//CONTINUE
		//GO_ROBOT:=LOADER_RS4_VAR.I_LOADER_RS4_READY_TAKEUP AND INPUT_G6_VAR.I_G6_READY_PLACING AND INDEXING_2_VAR.O_ROTATION_DONE AND INDEXING_1_VAR.I_INDEXING_1_ROTATION_DONE;
		IF LOADER_RS4_VAR.I_LOADER_RS4_READY_TAKEUP AND INPUT_G6_VAR.I_G6_READY_PLACING AND INDEXING_2_VAR.O_ROTATION_DONE AND INDEXING_1_VAR.I_INDEXING_1_ROTATION_DONE THEN
			GO_ROBOT:=TRUE;
		END_IF
		IF LOADER_RS4_VAR.I_LOADER_RS4_RUNNING AND GO_ROBOT AND NOT LOADER_RS4_VAR.I_LOADER_RS4_READY AND INDEXING_2_VAR.I_INDEXING_2_HOME AND INDEXING_2_VAR.O_ROTATION_DONE THEN
			//TMR3(IN:=GO_ROBOT,PT:=T#0.5S); 
			TMR3(IN:=TRUE,PT:=T#0.5S); 
			POSITION_CHANGED :=FALSE;
		ELSE
			TMR3(IN:=FALSE);
			INDEXING_1_VAR.O_ROTATION_START:=FALSE;	
		END_IF
		LOADER_RS4_VAR.O_LOADER_RS4_CONTINUE :=TMR3.q;
		IF TMR3.Q AND NOT LOADER_RS4_VAR.I_LOADER_RS4_END_CARRIER AND INDEXING_1_VAR.I_INDEXING_1_ROTATION_DONE AND INPUT_VAR.STRAIGHTEN_DONE AND INDEXING_2_VAR.I_INDEXING_2_HOME AND INDEXING_2_VAR.O_ROTATION_DONE  THEN
			IF LOADER_RS4_VAR.LOADER_RS4_OUTPUT_5 <=68  THEN
				POSITION_CHANGED :=TRUE;
			ELSE
				POSITION_CHANGED :=FALSE;
			END_IF	
		END_IF	

		IF ( LOADER_RS4_VAR.I_LOADER_RS4_READY_PLACING OR START_MOVE.Q OR GO_ROBOT)AND NOT LOADER_RS4_VAR.I_LOADER_RS4_READY THEN
			LOADER_RS4_VAR.O_LOADER_RS4_CONTINUE :=TRUE;
		ELSE
			LOADER_RS4_VAR.O_LOADER_RS4_CONTINUE :=FALSE;
		END_IF
	
//END CARRIER		
		IF LOADER_RS4_VAR.LOADER_RS4_OUTPUT_5 >=68 AND LOADER_RS4_VAR.I_LOADER_RS4_READY_TAKEUP THEN
			ROT_START(CLK:=TRUE);
			INDEXING_2_VAR.O_ROTATION_START:=ROT_START.Q;
			//LOADER_RS4_VAR.O_LOADER_RS4_STOP :=ROT_START.Q;
			 RESET_POSITION:=LOADER_RS4_VAR.I_LOADER_RS4_END_CARRIER;
			LOADER_RS4_VAR.I_LOADER_RS4_END_CARRIER:=TRUE;
			ELSE
			ROT_START(CLK:=FALSE);
		END_IF
		
		CNT_INC(CU:=LOADER_RS4_VAR.I_LOADER_RS4_READY_TAKEUP,RESET:= RESET_POSITION,PV:=17);
		LOADER_RS4_VAR.LOADER_RS4_OUTPUT_2:=(WORD_TO_BYTE(CNT_INC.CV)*4)+1 ;
		LOADER_RS4_VAR.LOADER_RS4_OUTPUT_3:=LOADER_RS4_VAR.LOADER_RS4_OUTPUT_2+1 ;
		LOADER_RS4_VAR.LOADER_RS4_OUTPUT_4:=LOADER_RS4_VAR.LOADER_RS4_OUTPUT_3+1 ;
		LOADER_RS4_VAR.LOADER_RS4_OUTPUT_5:=LOADER_RS4_VAR.LOADER_RS4_OUTPUT_4+1 ;
		START_MOVE (IN:=POSITION_CHANGED,PT:=T#0.1S);
	
		IF RESET_POSITION THEN
			RES_POS(IN:=RESET_POSITION,PT:=T#0.5S);
			LOADER_RS4_VAR.LOADER_RS4_OUTPUT_2:=1;
			LOADER_RS4_VAR.LOADER_RS4_OUTPUT_3:=2;
			LOADER_RS4_VAR.LOADER_RS4_OUTPUT_4:=3;
			LOADER_RS4_VAR.LOADER_RS4_OUTPUT_5:=4;
			IF RES_POS.Q THEN
				RESET_POSITION:=FALSE;
				RES_POS(IN:=FALSE);			
			END_IF
		END_IF
		IF NOT SORTER_RS4_VAR.I_SORTER_RS4_ENABLE THEN
			INDEXING_2_VAR.O_ROTATION_START:=LOADER_RS4_VAR.I_LOADER_RS4_END_CARRIER;
		END_IF
			
		CNT_CYCLE(CU:=INDEXING_2_VAR.O_ROTATION_DONE,RESET:=SORTER_RS4_VAR.I_SORTER_RS4_DISABLE,PV:=100);
		IF CNT_CYCLE.CV >=2 THEN
				IF INDEXING_2_VAR.O_ROTATION_DONE THEN
				SORTER_RS4_VAR.I_SORTER_RS4_ENABLE:=TRUE;
			END_IF
		END_IF
		
		IF LOADER_RS4_VAR.I_LOADER_RS4_START_PLACING AND INPUT_G6_VAR.I_G6_START_TAKEUP THEN
			INDEXING_1_VAR.O_ROTATION_START:=TRUE;
			
		END_IF
		IF LOADER_RS4_VAR.I_LOADER_RS4_READY_PLACING THEN
			GO_ROBOT:=FALSE;
		END_IF
		(*
		IF NOT CNT_CYCLE.Q AND LOADER_RS4_VAR.I_LOADER_RS4_END_CYCLE THEN
			START_ROTATE(CLK:=TRUE);
			INDEXING_2_VAR.O_ROTATION_START:= START_ROTATE.Q;	
			ELSE
			START_ROTATE(CLK:=FALSE);
		END_IF
					SORTER_RS4_VAR.I_SORTER_RS4_ENABLE:=TRUE;
		*)
	END_IF
END_IF


ELSE
	LOADER_RS4_VAR.O_LOADER_RS4_STOP:=TRUE;
	IF LOADER_RS4_VAR.I_LOADER_RS4_READY THEN
		LOADER_RS4_VAR.O_LOADER_RS4_SETMOTORON:=FALSE;
	END_IF
END_IF

END_PROGRAM

// ---- POUs/ROBOT/SORTER_RS4.TcPOU
PROGRAM SORTER_RS4
VAR

	TMR10: TON;
	TMR8: TON;
	TMR9: TON;
	TMR7: TON;
	TMR3: TON;
	POSITION_CHANGED: BOOL;
	START_MOVE: TP;
	TMR1: TON;
	TP2: TP;
	START_ROBOT: TP;
	TMR2: TON;
	GO_ROBOT: BOOL;
	TP_COUNT: R_TRIG;
	CNT_INC: CTU;
	VAL: INT;
	ROT_START:R_TRIG;
	RESET_POSITION: BOOL;
	RES_POS: TON;
	STRY_CONTINUE: TP;
END_VAR


IF SORTER_RS4_VAR.I_SORTER_RS4_ENABLE THEN
IF SORTER_RS4_VAR.IX_SORTER_RS4_GRIPPER_1 THEN
	SORTER_RS4_VAR.O_SORTER_RS4_GRIPPER_CLOSE_1:=TRUE;
	SORTER_RS4_VAR.O_SORTER_RS4_GRIPPER_OPEN_1:=FALSE;
ELSE
	SORTER_RS4_VAR.O_SORTER_RS4_GRIPPER_CLOSE_1:=FALSE;
	SORTER_RS4_VAR.O_SORTER_RS4_GRIPPER_OPEN_1:=TRUE;
END_IF

IF SORTER_RS4_VAR.IX_SORTER_RS4_GRIPPER_2 THEN
	SORTER_RS4_VAR.O_SORTER_RS4_GRIPPER_CLOSE_2:=TRUE;
	SORTER_RS4_VAR.O_SORTER_RS4_GRIPPER_OPEN_2:=FALSE;
ELSE
	SORTER_RS4_VAR.O_SORTER_RS4_GRIPPER_CLOSE_2:=FALSE;
	SORTER_RS4_VAR.O_SORTER_RS4_GRIPPER_OPEN_2:=TRUE;
END_IF

IF SORTER_RS4_VAR.IX_SORTER_RS4_GRIPPER_3 THEN
	SORTER_RS4_VAR.O_SORTER_RS4_GRIPPER_CLOSE_3:=TRUE;
	SORTER_RS4_VAR.O_SORTER_RS4_GRIPPER_OPEN_3:=FALSE;
ELSE
	SORTER_RS4_VAR.O_SORTER_RS4_GRIPPER_CLOSE_3:=FALSE;
	SORTER_RS4_VAR.O_SORTER_RS4_GRIPPER_OPEN_3:=TRUE;
END_IF

IF SORTER_RS4_VAR.IX_SORTER_RS4_GRIPPER_4 THEN
	SORTER_RS4_VAR.O_SORTER_RS4_GRIPPER_CLOSE_4:=TRUE;
	SORTER_RS4_VAR.O_SORTER_RS4_GRIPPER_OPEN_4:=FALSE;
ELSE
	SORTER_RS4_VAR.O_SORTER_RS4_GRIPPER_CLOSE_4:=FALSE;
	SORTER_RS4_VAR.O_SORTER_RS4_GRIPPER_OPEN_4:=TRUE;
END_IF

IF SORTER_RS4_VAR.IX_SORTER_RS4_GRIPPER_EXT_1 THEN
	SORTER_RS4_VAR.O_SORTER_RS4_GRIPPER_EXT_DOWN_1:=TRUE;
	SORTER_RS4_VAR.O_SORTER_RS4_GRIPPER_EXT_UP_1:=FALSE;
ELSE
	SORTER_RS4_VAR.O_SORTER_RS4_GRIPPER_EXT_DOWN_1:=FALSE;
	SORTER_RS4_VAR.O_SORTER_RS4_GRIPPER_EXT_UP_1:=TRUE;
END_IF


IF SORTER_RS4_VAR.IX_SORTER_RS4_GRIPPER_EXT_2 THEN
	SORTER_RS4_VAR.O_SORTER_RS4_GRIPPER_EXT_DOWN_2:=TRUE;
	SORTER_RS4_VAR.O_SORTER_RS4_GRIPPER_EXT_UP_2:=FALSE;
ELSE
	SORTER_RS4_VAR.O_SORTER_RS4_GRIPPER_EXT_DOWN_2:=FALSE;
	SORTER_RS4_VAR.O_SORTER_RS4_GRIPPER_EXT_UP_2:=TRUE;
END_IF


IF SORTER_RS4_VAR.IX_SORTER_RS4_GRIPPER_EXT_3 THEN
	SORTER_RS4_VAR.O_SORTER_RS4_GRIPPER_EXT_DOWN_3:=TRUE;
	SORTER_RS4_VAR.O_SORTER_RS4_GRIPPER_EXT_UP_3:=FALSE;
ELSE
	SORTER_RS4_VAR.O_SORTER_RS4_GRIPPER_EXT_DOWN_3:=FALSE;
	SORTER_RS4_VAR.O_SORTER_RS4_GRIPPER_EXT_UP_3:=TRUE;
END_IF


IF SORTER_RS4_VAR.IX_SORTER_RS4_GRIPPER_EXT_4 THEN
	SORTER_RS4_VAR.O_SORTER_RS4_GRIPPER_EXT_DOWN_4:=TRUE;
	SORTER_RS4_VAR.O_SORTER_RS4_GRIPPER_EXT_UP_4:=FALSE;
ELSE
	SORTER_RS4_VAR.O_SORTER_RS4_GRIPPER_EXT_DOWN_4:=FALSE;
	SORTER_RS4_VAR.O_SORTER_RS4_GRIPPER_EXT_UP_4:=TRUE;
END_IF


SORTER_RS4_VAR.O_SORTER_RS4_SETMOTORON:=TRUE;
TMR1(IN:=SORTER_RS4_VAR.O_SORTER_RS4_SETMOTORON ,PT:=T#0.5S);
IF TMR1.Q THEN
	TP2(IN:=TMR1.Q,PT:=T#1S);
	SORTER_RS4_VAR.O_SORTER_RS4_STOP:=TP2.Q;
END_IF
IF SORTER_RS4_VAR.O_SORTER_RS4_SETMOTORON AND INDEXING_2_VAR.I_INDEXING_2_ROTATION_DONE AND INDEXING_2_VAR.I_INDEXING_2_HOME THEN
	IF SORTER_RS4_VAR.I_SORTER_RS4_READY OR SORTER_RS4_VAR.I_SORTER_RS4_RUNNING THEN
//ERROR OVERRIDE
		IF SORTER_RS4_VAR.I_SORTER_RS4_ERROR THEN
			TMR10(IN:=SORTER_RS4_VAR.I_SORTER_RS4_ERROR,PT:=T#1S);
			IF TMR10.Q THEN
				SORTER_RS4_VAR.O_SORTER_RS4_RESET :=TRUE;	
			ELSE
				SORTER_RS4_VAR.O_SORTER_RS4_RESET :=FALSE;
			END_IF
		END_IF 

//START FOR 1ST TIME			
		IF SORTER_RS4_VAR.I_SORTER_RS4_READY AND NOT SORTER_RS4_VAR.I_SORTER_RS4_ERROR AND NOT SORTER_RS4_VAR.I_SORTER_RS4_RUNNING THEN
			TMR7(IN:=INDEXING_2_VAR.I_INDEXING_2_ROTATION_DONE,PT:=T#1S);
			START_ROBOT(IN:=TMR7.Q,PT:=T#3S);
			SORTER_RS4_VAR.O_SORTER_RS4_START :=TMR7.Q;
			RESET_POSITION:=TRUE;
		ELSE
			TMR7(IN:=FALSE);
		END_IF
			IF SORTER_RS4_VAR.I_SORTER_RS4_RUNNING AND SORTER_RS4_VAR.I_SORTER_RS4_READY_TAKEUP THEN
			SORTER_RS4_VAR.O_SORTER_RS4_START :=FALSE ;
		END_IF
		
		//STOP
		IF SORTER_RS4_VAR.I_SORTER_RS4_END_CARRIER AND NOT SORTER_RS4_VAR.I_SORTER_RS4_READY AND NOT SORTER_RS4_VAR.I_SORTER_RS4_RUNNING THEN
			TMR8(IN:=FALSE);
			TMR9(IN:=FALSE);
			SORTER_RS4_VAR.O_SORTER_RS4_STOP :=TRUE;
		END_IF
			TMR2(IN:=SORTER_RS4_VAR.O_SORTER_RS4_STOP,PT:=T#1S);
		IF TMR2.Q THEN
			SORTER_RS4_VAR.I_SORTER_RS4_HANG:=FALSE;
			SORTER_RS4_VAR.O_SORTER_RS4_STOP:=FALSE;
			TMR1(IN:=FALSE);
		END_IF	
			
//CONTINUE
		GO_ROBOT:=(SORTER_RS4_VAR.I_SORTER_RS4_READY_TAKEUP AND LOADER_RS4_VAR.I_LOADER_RS4_START_PLACING)  AND INDEXING_2_VAR.O_ROTATION_DONE ;
		IF SORTER_RS4_VAR.I_SORTER_RS4_RUNNING AND  GO_ROBOT AND NOT SORTER_RS4_VAR.I_SORTER_RS4_READY AND INDEXING_2_VAR.I_INDEXING_2_HOME AND INDEXING_2_VAR.O_ROTATION_DONE THEN
			TMR3(IN:=GO_ROBOT,PT:=T#0.5S); 
			POSITION_CHANGED :=FALSE;
		ELSE
			TMR3(IN:=FALSE);
			INDEXING_2_VAR.O_ROTATION_START:=FALSE;	
		END_IF

		IF TMR3.Q AND NOT SORTER_RS4_VAR.I_SORTER_RS4_END_CARRIER AND INDEXING_2_VAR.I_INDEXING_2_ROTATION_DONE AND INPUT_VAR.STRAIGHTEN_DONE AND INDEXING_2_VAR.I_INDEXING_2_HOME  THEN
			IF SORTER_RS4_VAR.SORTER_RS4_POS_TAKEUP_4 <=68  THEN
				POSITION_CHANGED :=TRUE;
			ELSE
				POSITION_CHANGED :=FALSE;
				
			END_IF	
		END_IF	

		IF  START_MOVE.Q AND NOT SORTER_RS4_VAR.I_SORTER_RS4_READY OR STRY_CONTINUE.Q OR SORTER_RS4_VAR.I_SORTER_RS4_READY_PLACING THEN
			SORTER_RS4_VAR.O_SORTER_RS4_CONTINUE :=TRUE;
		ELSE
			SORTER_RS4_VAR.O_SORTER_RS4_CONTINUE :=FALSE;
		END_IF
	
//END CARRIER		
		IF SORTER_RS4_VAR.SORTER_RS4_POS_TAKEUP_4 >=68 AND SORTER_RS4_VAR.I_SORTER_RS4_READY_takeup THEN
			ROT_START(CLK:=TRUE);
			//INDEXING_2_VAR.O_ROTATION_START:=ROT_START.Q;
			 RESET_POSITION:=SORTER_RS4_VAR.I_SORTER_RS4_END_CARRIER;
			SORTER_RS4_VAR.I_SORTER_RS4_END_CARRIER:=TRUE;
			ELSE
			ROT_START(CLK:=FALSE);
		END_IF
		
//POSITION TAKE UP		
		CNT_INC(CU:=SORTER_RS4_VAR.I_SORTER_RS4_START_PLACING,RESET:= ROT_START.Q,PV:=17);
		SORTER_RS4_VAR.SORTER_RS4_POS_TAKEUP_1:=(WORD_TO_BYTE(CNT_INC.CV)*4)+1 ;
		SORTER_RS4_VAR.SORTER_RS4_POS_TAKEUP_2:=SORTER_RS4_VAR.SORTER_RS4_POS_TAKEUP_1+1 ;
		SORTER_RS4_VAR.SORTER_RS4_POS_TAKEUP_3:=SORTER_RS4_VAR.SORTER_RS4_POS_TAKEUP_2+1 ;
		SORTER_RS4_VAR.SORTER_RS4_POS_TAKEUP_4:=SORTER_RS4_VAR.SORTER_RS4_POS_TAKEUP_3+1 ;
		START_MOVE (IN:=POSITION_CHANGED,PT:=T#0.1S);
		
//SORTER_RS4_POS_TAKEUP_1
		IF RESET_POSITION THEN
			RES_POS(IN:=RESET_POSITION,PT:=T#0.5S);
			SORTER_RS4_VAR.SORTER_RS4_POS_TAKEUP_1:=1;
			SORTER_RS4_VAR.SORTER_RS4_POS_TAKEUP_2:=2;
			SORTER_RS4_VAR.SORTER_RS4_POS_TAKEUP_3:=3;
			SORTER_RS4_VAR.SORTER_RS4_POS_TAKEUP_4:=4;
			IF RES_POS.Q THEN
				RESET_POSITION:=FALSE;
				RES_POS(IN:=FALSE);			
			END_IF
		END_IF
		
		STRY_CONTINUE(IN:=SORTER_RS4_VAR.I_SORTER_RS4_RUNNING,PT:=T#2S);
	END_IF
END_IF


ELSE
	SORTER_RS4_VAR.O_SORTER_RS4_STOP:=TRUE;
	IF SORTER_RS4_VAR.I_SORTER_RS4_READY THEN
		SORTER_RS4_VAR.O_SORTER_RS4_SETMOTORON:=FALSE;
	END_IF
END_IF

END_PROGRAM

// ---- POUs/LOADER/STRAIGHTENING_PROG_1.TcPOU
 PROGRAM STRAIGHTENING_PROG_1
VAR

	NEW: INT;
	FG: INT;
	ENABLE_TIMER: BOOL := FALSE;
	TMR1: TON;
	TMR2: TON;
	CNT1: CTU;
END_VAR

IF INPUT_VAR.STRAIGHTEN_START AND INDEXING_1_VAR.I_INDEXING_1_ROTATION_DONE THEN
	ENABLE_TIMER:=TRUE;
END_IF
IF ENABLE_TIMER THEN
	INPUT_VAR.STRAIGHTEN_START:=FALSE;
	TMR1(IN:=NOT TMR2.Q,PT:=T#0.07S);
	TMR2(IN:=TMR1.Q,PT:=T#0.15S);
	IF TMR2.Q THEN
		TMR1(IN:=FALSE); 
		TMR2(IN:=FALSE);
	END_IF
	
	IF NOT  INDEXING_1_VAR.I_PRESS_STOPPER_DOWN  THEN
		INDEXING_1_VAR.O_PRESS_STOPPER_DOWN:=TRUE;
		INDEXING_1_VAR.O_PRESS_STOPPER_UP:=FALSE;
	END_IF
ELSE
		TMR1(IN:=FALSE);
		TMR2(IN:=FALSE);
END_IF

CNT1(CU:=TMR1.Q,RESET:=NOT	ENABLE_TIMER,PV:=5);
IF CNT1.CV >=10 THEN
	ENABLE_TIMER:=FALSE;
	INDEXING_1_VAR.STRAIGHTEN_FINISH:=TRUE;
	INDEXING_1_VAR.O_PRESS_STOPPER_DOWN:=FALSE;
	INDEXING_1_VAR.O_PRESS_STOPPER_UP:=TRUE;
END_IF

IF CNT1.CV =2 THEN
	INDEXING_1_VAR.STRAIGHTEN_FINISH:=FALSE;
END_IF

IF 	INDEXING_1_VAR.STRAIGHTEN_FINISH THEN
	IF INDEXING_1_VAR.I_PRESS_STOPPER_UP THEN
		INPUT_VAR.STRAIGHTEN_DONE :=TRUE;	
		INPUT_VAR.STRAIGHTEN_PROCESS:=FALSE;
	END_IF	
END_IF
CASE CNT1.CV OF	
//CASE INDEXING_1_VAR.INDEXING_1_CASE OF
0:	
	INDEXING_1_VAR.O_PRESS_STOPPER_DOWN:=FALSE;
	INDEXING_1_VAR.O_PRESS_STOPPER_UP:=TRUE;
	//INDEXING_1_VAR.I_INDEXING_1_ROTATION_DONE:=FALSE;
	INDEXING_1_VAR.I_INDEXING_1_READY_FOR_STRAIGHTEN:=FALSE;
1:	
	INPUT_VAR.STRAIGHTEN_PROCESS:=TRUE;
	INDEXING_1_VAR.O_INDEXING_1_GRIPPER_OPEN_1:=TRUE;
	INDEXING_1_VAR.O_INDEXING_1_GRIPPER_CLOSE_1:=FALSE;
		
2:
	INDEXING_1_VAR.O_INDEXING_1_GRIPPER_EXT_UP :=TRUE;	
	INDEXING_1_VAR.O_INDEXING_1_GRIPPER_EXT_down:=FALSE;

		
3:
	INDEXING_1_VAR.O_INDEXING_1_GRIPPER_OPEN_1:=FALSE;
	INDEXING_1_VAR.O_INDEXING_1_GRIPPER_CLOSE_1:=TRUE;
			
4:
	INDEXING_1_VAR.O_INDEXING_1_GRIPPER_EXT_UP :=FALSE;	
	INDEXING_1_VAR.O_INDEXING_1_GRIPPER_EXT_down:=TRUE;

5:	
	INDEXING_1_VAR.O_INDEXING_1_GRIPPER_OPEN_1:=TRUE;
	INDEXING_1_VAR.O_INDEXING_1_GRIPPER_CLOSE_1:=FALSE;
		
6:
	INDEXING_1_VAR.O_INDEXING_1_GRIPPER_EXT_UP :=TRUE;	
	INDEXING_1_VAR.O_INDEXING_1_GRIPPER_EXT_down:=FALSE;	
7:
	INDEXING_1_VAR.O_INDEXING_1_GRIPPER_OPEN_1:=FALSE;
	INDEXING_1_VAR.O_INDEXING_1_GRIPPER_CLOSE_1:=TRUE;
			
8:
	INDEXING_1_VAR.O_INDEXING_1_GRIPPER_EXT_UP :=FALSE;	
	INDEXING_1_VAR.O_INDEXING_1_GRIPPER_EXT_down:=TRUE;

END_CASE

IF 
	INDEXING_1_VAR.O_INDEXING_1_GRIPPER_OPEN_1 AND
	INDEXING_1_VAR.I_INDEXING_1_GRIPPER_OPEN_1 AND
	INDEXING_1_VAR.I_INDEXING_1_GRIPPER_OPEN_2	AND
	INDEXING_1_VAR.I_INDEXING_1_GRIPPER_OPEN_3	AND 
	INDEXING_1_VAR.I_INDEXING_1_GRIPPER_OPEN_4	AND
	NOT INDEXING_1_VAR.I_INDEXING_1_GRIPPER_CLOSE_1	AND
	NOT INDEXING_1_VAR.I_INDEXING_1_GRIPPER_CLOSE_2	AND
	NOT INDEXING_1_VAR.I_INDEXING_1_GRIPPER_CLOSE_3	AND
	NOT INDEXING_1_VAR.I_INDEXING_1_GRIPPER_CLOSE_4 THEN
		INDEXING_1_VAR.I_ALL_GRIPPER_OPEN :=TRUE;
	END_IF

IF 
	NOT INDEXING_1_VAR.O_INDEXING_1_GRIPPER_OPEN_1 AND
	NOT INDEXING_1_VAR.I_INDEXING_1_GRIPPER_OPEN_1 AND
	NOT INDEXING_1_VAR.I_INDEXING_1_GRIPPER_OPEN_2	AND
	NOT INDEXING_1_VAR.I_INDEXING_1_GRIPPER_OPEN_3	AND 
	NOT INDEXING_1_VAR.I_INDEXING_1_GRIPPER_OPEN_4	AND
	INDEXING_1_VAR.I_INDEXING_1_GRIPPER_CLOSE_1	AND
	INDEXING_1_VAR.I_INDEXING_1_GRIPPER_CLOSE_2	AND
	INDEXING_1_VAR.I_INDEXING_1_GRIPPER_CLOSE_3	AND
	INDEXING_1_VAR.I_INDEXING_1_GRIPPER_CLOSE_4 THEN
		INDEXING_1_VAR.I_ALL_GRIPPER_OPEN :=FALSE;
END_IF


	INDEXING_1_VAR.O_INDEXING_1_GRIPPER_OPEN_2:=INDEXING_1_VAR.O_INDEXING_1_GRIPPER_OPEN_1;
	INDEXING_1_VAR.O_INDEXING_1_GRIPPER_OPEN_3:=INDEXING_1_VAR.O_INDEXING_1_GRIPPER_OPEN_1;
	INDEXING_1_VAR.O_INDEXING_1_GRIPPER_OPEN_4:=INDEXING_1_VAR.O_INDEXING_1_GRIPPER_OPEN_1;

	INDEXING_1_VAR.O_INDEXING_1_GRIPPER_CLOSE_2:=INDEXING_1_VAR.O_INDEXING_1_GRIPPER_CLOSE_1;
	INDEXING_1_VAR.O_INDEXING_1_GRIPPER_CLOSE_3:=INDEXING_1_VAR.O_INDEXING_1_GRIPPER_CLOSE_1;
	INDEXING_1_VAR.O_INDEXING_1_GRIPPER_CLOSE_4:=INDEXING_1_VAR.O_INDEXING_1_GRIPPER_CLOSE_1;

END_PROGRAM

// ---- POUs/LASER/LOAD_LASER.TcPOU
PROGRAM LOAD_LASER
VAR_INPUT

END_VAR

VAR
	TMR_DELAY: TON;
	TMR1:TON;
	TMR_STOPPER_A: TON;
	TMR_STOPPER_B: TON;
END_VAR

CASE SORTER_VAR.I_CASE OF
0: //standby near lotbox
	IF SORTER_VAR.ACTIVE_ID=6 THEN
		SORTER_VAR.ACTIVE_ID:=1;
	END_IF
	CASE SORTER_VAR.I_CURRENT_TRANSACTION.TRANSPORT_INDEX OF
		2 : LASER_MOVE(STEP_DATA_1:=SORTER_VAR.I_CURRENT_TRANSACTION.STATION_NUMBER_LOAD,
				STEP_DATA_2:=3,
				STEP_DATA_3:=SORTER_VAR.I_CURRENT_TRANSACTION.JIG_INDEX_LOAD,
				STEP_DATA_4:=0,
				STEP_DATA_5:=1);
				SORTER_VAR.O_STOPPER_TRANSFER_B:=FALSE;
		1 : LASER_MOVE(STEP_DATA_1:=SORTER_VAR.I_CURRENT_TRANSACTION.STATION_NUMBER_LOAD,
				STEP_DATA_2:=3,
				STEP_DATA_3:=SORTER_VAR.I_CURRENT_TRANSACTION.JIG_INDEX_LOAD,
				STEP_DATA_4:=1,
				STEP_DATA_5:=0);
				SORTER_VAR.O_STOPPER_TRANSFER_A:=FALSE;
	END_CASE			
	SORTER_VAR.O_VACUUM_On:=FALSE;
	SORTER_VAR.O_VACUUM_OFF:=FALSE;	
	
			
1: //standby near lotbox
	
	IF SORTER_VAR.ACTIVE_ID=6 THEN
		SORTER_VAR.ACTIVE_ID:=1;
	END_IF
		LASER_MOVE(STEP_DATA_1:=SORTER_VAR.I_CURRENT_TRANSACTION.STATION_NUMBER_LOAD,
				STEP_DATA_2:=4,
				STEP_DATA_3:=SORTER_VAR.I_CURRENT_TRANSACTION.JIG_INDEX_LOAD,
				STEP_DATA_4:=0,
				STEP_DATA_5:=0);

		CASE SORTER_VAR.I_CURRENT_TRANSACTION.TRANSPORT_INDEX OF
		1:
			SORTER_VAR.I_LOADING_DONE_A:=FALSE;
		
		2:
			SORTER_VAR.I_LOADING_DONE_B:=FALSE;
	END_CASE
	
				
2://vacuum position 
	IF SORTER_VAR.ACTIVE_ID=6 THEN
		SORTER_VAR.ACTIVE_ID:=1;
	END_IF
	SORTER_VAR.I_CASE:=SORTER_VAR.I_CASE+1;
	(*LASER_MOVE(STEP_DATA_1:=SORTER_VAR.I_CURRENT_TRANSACTION.STATION_NUMBER_LOAD,
				STEP_DATA_2:=4,
				STEP_DATA_3:=SORTER_VAR.I_CURRENT_TRANSACTION.JIG_INDEX_LOAD,
				STEP_DATA_4:=0,
				STEP_DATA_5:=0);
	IF SORTER_VAR.ACTIVE_ID=3 THEN
		SORTER_VAR.O_VACUUM_ON:=TRUE;
		SORTER_VAR.O_VACUUM_OFF:=FALSE;	
	END_IF
	*)

3://vacuum position 
	IF SORTER_VAR.ACTIVE_ID=6 THEN
		SORTER_VAR.ACTIVE_ID:=1; 
	END_IF
	SORTER_VAR.I_CASE:=SORTER_VAR.I_CASE+1;
(*
		LASER_MOVE(STEP_DATA_1:=SORTER_VAR.I_CURRENT_TRANSACTION.STATION_NUMBER_LOAD,
				STEP_DATA_2:=4,
				STEP_DATA_3:=SORTER_VAR.I_CURRENT_TRANSACTION.JIG_INDEX_LOAD,
				STEP_DATA_4:=0,
				STEP_DATA_5:=0);
*)
4://vacuum position 
	IF SORTER_VAR.ACTIVE_ID=6 THEN
		SORTER_VAR.ACTIVE_ID:=1;
	END_IF
	SORTER_VAR.O_VACUUM_ON:=TRUE;
	SORTER_VAR.O_VACUUM_OFF:=FALSE;
	//CHECK JIG LASER PRESENCE	
LASER_MOVE(STEP_DATA_1:=SORTER_VAR.I_CURRENT_TRANSACTION.STATION_NUMBER_LOAD,
				STEP_DATA_2:=4,
				STEP_DATA_3:=SORTER_VAR.I_CURRENT_TRANSACTION.JIG_INDEX_LOAD,
				STEP_DATA_4:=0,
				STEP_DATA_5:=0);
(*		
	IF  SORTER_VAR.O_VACUUM_ON THEN
		TMR1(IN:=TRUE,PT:=T#2S);
		IF TMR1.Q THEN
			IF  SORTER_VAR.I_VACUUM_ON AND SORTER_VAR.O_VACUUM_ON THEN
				SORTER_VAR.JIG_LASER_PRESENCE :=TRUE;
				
				LASER_MOVE(STEP_DATA_1:=7,
				STEP_DATA_2:=4,
				STEP_DATA_3:=SORTER_VAR.I_CURRENT_TRANSACTION.JIG_INDEX_LOAD,
				STEP_DATA_4:=0,
				STEP_DATA_5:=0);
			ELSE
				SORTER_VAR.JIG_LASER_PRESENCE :=FALSE;	
				LASER_MOVE(STEP_DATA_1:=SORTER_VAR.I_CURRENT_TRANSACTION.STATION_NUMBER_LOAD,
				STEP_DATA_2:=2,
				STEP_DATA_3:=SORTER_VAR.I_CURRENT_TRANSACTION.JIG_INDEX_LOAD,
				STEP_DATA_4:=0,
				STEP_DATA_5:=0);
				
				LASER_MOVE(STEP_DATA_1:=SORTER_VAR.I_CURRENT_TRANSACTION.STATION_NUMBER_LOAD,
				STEP_DATA_2:=1,
				STEP_DATA_3:=SORTER_VAR.I_CURRENT_TRANSACTION.JIG_INDEX_LOAD,
				STEP_DATA_4:=0,
				STEP_DATA_5:=0);
				
				TMR_DELAY(IN:=TRUE,PT:=T#2S);
				IF TMR_DELAY.Q THEN
					FLAG_VAR.ALLOW_EXECUTE_LOAD_LASER:=FALSE;
					SORTER_VAR.I_CURRENT_TRANSACTION.JIG_INDEX_LOAD:=SORTER_VAR.I_CURRENT_TRANSACTION.JIG_INDEX_LOAD+0;
					SORTER_VAR.I_CASE:=0;
					TMR1(IN:=FALSE);
					SORTER_VAR.O_VACUUM_ON:=FALSE;
					SORTER_VAR.O_VACUUM_OFF:=FALSE;
				END_IF
			END_IF
		END_IF 
	END_IF
*)
				

5://vacuum position 
	IF SORTER_VAR.ACTIVE_ID=6 THEN
		SORTER_VAR.ACTIVE_ID:=1;
	END_IF

	LASER_MOVE(STEP_DATA_1:=SORTER_VAR.I_CURRENT_TRANSACTION.STATION_NUMBER_LOAD,//9,
				STEP_DATA_2:=2,
				STEP_DATA_3:=SORTER_VAR.I_CURRENT_TRANSACTION.JIG_INDEX_LOAD,
				STEP_DATA_4:=0,
				STEP_DATA_5:=0);

6://gripping position
	IF SORTER_VAR.ACTIVE_ID=6 THEN
		SORTER_VAR.ACTIVE_ID:=1;
	END_IF

	LASER_MOVE(STEP_DATA_1:=SORTER_VAR.I_CURRENT_TRANSACTION.TRANSPORT_INDEX+5,
				STEP_DATA_2:=1,
				STEP_DATA_3:=12,
				STEP_DATA_4:=0,
				STEP_DATA_5:=0);


7://placing onto LASER transport
	IF SORTER_VAR.ACTIVE_ID=6 THEN
		SORTER_VAR.ACTIVE_ID:=1;
	END_IF
	LASER_MOVE(STEP_DATA_1:=SORTER_VAR.I_CURRENT_TRANSACTION.TRANSPORT_INDEX+5,
				STEP_DATA_2:=1,
				STEP_DATA_3:=11,
				STEP_DATA_4:=0,
				STEP_DATA_5:=0);

8://placing onto LASER transport
	IF SORTER_VAR.ACTIVE_ID=6 THEN
		SORTER_VAR.ACTIVE_ID:=1;
	END_IF
	
	LASER_MOVE(STEP_DATA_1:=SORTER_VAR.I_CURRENT_TRANSACTION.TRANSPORT_INDEX+5,
				STEP_DATA_2:=1,
				STEP_DATA_3:=11,
				STEP_DATA_4:=0,
				STEP_DATA_5:=0);
	(*IF SORTER_VAR.ACTIVE_ID=3 THEN
		SORTER_VAR.O_VACUUM_On:=FALSE;
		SORTER_VAR.O_VACUUM_OFF:=TRUE;	
	END_IF
	*)
	
9://homing
	IF SORTER_VAR.ACTIVE_ID=6 THEN
		SORTER_VAR.ACTIVE_ID:=1;
	END_IF
	
			LASER_MOVE(STEP_DATA_1:=SORTER_VAR.I_CURRENT_TRANSACTION.TRANSPORT_INDEX+5,
				STEP_DATA_2:=0,
				STEP_DATA_3:=11,
				STEP_DATA_4:=0,
				STEP_DATA_5:=0);
	(*
	IF SORTER_VAR.I_VACUUM_ON THEN
		LASER_MOVE(STEP_DATA_1:=SORTER_VAR.I_CURRENT_TRANSACTION.TRANSPORT_INDEX+5,
				STEP_DATA_2:=1,
				STEP_DATA_3:=11,
				STEP_DATA_4:=0,
				STEP_DATA_5:=0);
	ELSE
		SORTER_VAR.O_VACUUM_On:=FALSE;
		SORTER_VAR.O_VACUUM_OFF:=TRUE;
	END_IF	
	*)			
10://pusH LASER transport
	IF SORTER_VAR.ACTIVE_ID=6 THEN
		SORTER_VAR.ACTIVE_ID:=1;
	END_IF
	SORTER_VAR.O_VACUUM_OFF:=FALSE;
	CASE SORTER_VAR.I_CURRENT_TRANSACTION.TRANSPORT_INDEX OF
		2 :
			IF NOT SORTER_VAR.I_LASER_TRANSFER_AT_FRONT_B THEN
				LASER_MOVE(STEP_DATA_1:=0,
				STEP_DATA_2:=0,
				STEP_DATA_3:=0,
				STEP_DATA_4:=0,
				STEP_DATA_5:=2);
			END_IF
				 
		1 : 
			IF NOT SORTER_VAR.I_LASER_TRANSFER_AT_FRONT_A THEN
				LASER_MOVE(STEP_DATA_1:=0,
				STEP_DATA_2:=0,
				STEP_DATA_3:=0,
				STEP_DATA_4:=2,
				STEP_DATA_5:=0);
			END_IF
	END_CASE			 
11:
				CASE SORTER_VAR.I_CURRENT_TRANSACTION.TRANSPORT_INDEX OF
		1:	
			//IF SORTER_VAR.I_LASER_TRANSFER_AT_FRONT_A THEN
				
				TMR_STOPPER_A(IN:=TRUE,PT:=T#0.8S);
				IF TMR_STOPPER_A.Q THEN
					SORTER_VAR.O_STOPPER_TRANSFER_A:=TRUE;
					SORTER_VAR.I_LOADING_DONE_A:=TRUE;
					TMR1(IN:=FALSE);
	TMR_DELAY(IN:=FALSE);
	FLAG_VAR.ALLOW_EXECUTE_LOAD_LASER:=FALSE;	
					SORTER_VAR.I_CASE:=100;
						SORTER_VAR.O_VACUUM_On:=FALSE;
	SORTER_VAR.O_VACUUM_OFF:=FALSE;
	
END_IF
				
(*			ELSE
				TMR_STOPPER_A(IN:=FALSE);
				LASER_MOVE(STEP_DATA_1:=0,
				STEP_DATA_2:=0,
				STEP_DATA_3:=0,
				STEP_DATA_4:=2,
				STEP_DATA_5:=0);
			END_IF
*)			
			2:
			//IF SORTER_VAR.I_LASER_TRANSFER_AT_FRONT_B THEN
				
				TMR_STOPPER_B(IN:=TRUE,PT:=T#0.8S);
				IF TMR_STOPPER_B.Q THEN
					SORTER_VAR.O_STOPPER_TRANSFER_B:=TRUE;	
					SORTER_VAR.I_LOADING_DONE_B:=TRUE;
					TMR1(IN:=FALSE);
	TMR_DELAY(IN:=FALSE);
	FLAG_VAR.ALLOW_EXECUTE_LOAD_LASER:=FALSE;	
					SORTER_VAR.I_CASE:=100;
						SORTER_VAR.O_VACUUM_On:=FALSE;
	SORTER_VAR.O_VACUUM_OFF:=FALSE;
			END_IF
(*			ELSE
				TMR_STOPPER_B(IN:=FALSE);
				LASER_MOVE(STEP_DATA_1:=0,
				STEP_DATA_2:=0,
				STEP_DATA_3:=0,
				STEP_DATA_4:=0,
				STEP_DATA_5:=2);
			END_IF
*)			
	END_CASE
100:
	SORTER_VAR.O_VACUUM_On:=FALSE;
	SORTER_VAR.O_VACUUM_OFF:=FALSE;
	TMR1(IN:=FALSE);
	TMR_DELAY(IN:=FALSE);
	FLAG_VAR.ALLOW_EXECUTE_LOAD_LASER:=FALSE;								
								
END_CASE

END_PROGRAM

// ---- POUs/LASER/LASER_MOVE.TcPOU
PROGRAM LASER_MOVE
//FUNCTION LASER_MOVE : BOOL
VAR_INPUT
	STEP_DATA_1: BYTE;
	STEP_DATA_2: BYTE;
	STEP_DATA_3: BYTE;
	STEP_DATA_4: BYTE;
	STEP_DATA_5: BYTE;

END_VAR

VAR
	
	(*
DataWordInput1 AT %IB232 : ARRAY [0..15] OF WORD; 
DataWordInput2 AT %IB264 : ARRAY [16..31] OF WORD;
DataWordInput3 AT %IB264 : ARRAY [32..47] OF WORD; 
DataWordInput4 AT %IB296 : ARRAY [48..56] OF WORD; 
DataWordOutput1 AT %QB232 : ARRAY [0..15] OF WORD; 
DataWordOutput2 AT %QB264 : ARRAY [16..31] OF WORD; 
DataWordOutput3 AT %QB296 : ARRAY [32..47] OF WORD; 
DataWordOutput4 AT %QB328 : ARRAY [48..56] OF WORD; 

DataWordInput1 AT %IB100 : ARRAY [0..15] OF WORD; 
DataWordInput2 AT %IB132 : ARRAY [16..31] OF WORD; 
DataWordInput3 AT %IB164 : ARRAY [32..47] OF WORD; 
DataWordInput4 AT %IB196 : ARRAY [48..56] OF WORD; 
DataWordOutput1 AT %QB100 : ARRAY [0..15] OF WORD; 
DataWordOutput2 AT %QB132 : ARRAY [16..31] OF WORD; 
DataWordOutput3 AT %QB164 : ARRAY [32..47] OF WORD; 
DataWordOutput4 AT %QB196 : ARRAY [48..56] OF WORD; 
	*)
	Gateway_Q0_MODE_COMMAND_0 AT %QX232.0 : BOOL ;
	Gateway_Q0_MODE_COMMAND_1 AT %QX232.1 : BOOL ;
	Gateway_Q0_RESET AT %QX232.4 : BOOL;
	Gateway_Q0_RESTART AT %QX232.5 : BOOL;
	Gateway_Q0_STOP AT %QX232.7 : BOOL;
	Gateway_Q1_0 AT %QX233.0 : BOOL;
	Gateway_Q1_1 AT %QX233.1 : BOOL;
	Gateway_Q1_2 AT %QX233.2 : BOOL;
	Gateway_Q1_3 AT %QX233.3 : BOOL;
	Gateway_Q1_4 AT %QX233.4 : BOOL;
	Gateway_Gateway_Unit_2_Status AT %QB234 : BYTE;
	Gateway_Q3_0 AT %QX235.0 : BOOL;
	Gateway_Q3_1 AT %QX235.1 : BOOL;
	Gateway_Q3_2 AT %QX235.2 : BOOL;
	Gateway_Q3_3 AT %QX235.3 : BOOL;	
	

	ID1_StepData AT %QB246 : BYTE;
	ID1_Hold AT %QX247.0 : BOOL;
	ID1_SVON AT %QX247.1 : BOOL;
	ID1_Drive AT %QX247.2 : BOOL;
	ID1_Reset AT %QX247.3 : BOOL;
	ID1_Setup AT %QX247.4 : BOOL;
	

	ID2_StepData AT %QB266 : BYTE;
	ID2_Hold AT %QX267.0 : BOOL;
	ID2_SVON AT %QX267.1 : BOOL;
	ID2_Drive AT %QX267.2 : BOOL;
	ID2_Reset AT %QX267.3 : BOOL;
	ID2_Setup AT %QX267.4 : BOOL;


	ID3_StepData AT %QB286 : BYTE;
	ID3_Hold AT %QX287.0 : BOOL;
	ID3_SVON AT %QX287.1 : BOOL;
	ID3_Drive AT %QX287.2 : BOOL;
	ID3_Reset AT %QX287.3 : BOOL;
	ID3_Setup AT %QX287.4 : BOOL;
	
	
	ID4_StepData AT %QB306 : BYTE;
	ID4_Hold AT %QX307.0 : BOOL;
	ID4_SVON AT %QX307.1 : BOOL;
	ID4_Drive AT %QX307.2 : BOOL;
	ID4_Reset AT %QX307.3 : BOOL;
	ID4_Setup AT %QX307.4 : BOOL;
	

	ID5_StepData AT %QB326 : BYTE;
	ID5_Hold AT %QX327.0 : BOOL;
	ID5_SVON AT %QX327.1 : BOOL;
	ID5_Drive AT %QX327.2 : BOOL;
	ID5_Reset AT %QX327.3 : BOOL;
	ID5_Setup AT %QX327.4 : BOOL;
	
	byte0 : BYTE;
	byte1 : BYTE;
	byte2 : BYTE;
	byte3 : BYTE;
	
	bit14_0 : BOOL;
	bit14_1 : BOOL;
	bit14_2 : BOOL;
	bit14_3 : BOOL;
	bit14_4 : BOOL;
	bit14_5 : BOOL;
	
	bit15_0 : BOOL;
	bit15_1 : BOOL;
	bit15_2 : BOOL;
	bit15_3 : BOOL;
	bit15_4 : BOOL; 
	
	bit34_0 : BOOL;
	bit34_1 : BOOL;
	bit34_2 : BOOL;
	bit34_3 : BOOL;
	bit34_4 : BOOL;
	bit34_5 : BOOL;
	
	bit35_0 : BOOL;
	bit35_1 : BOOL;
	bit35_2 : BOOL;
	bit35_3 : BOOL;
	bit35_4 : BOOL; 
	
	bit54_0 : BOOL;
	bit54_1 : BOOL;
	bit54_2 : BOOL;
	bit54_3 : BOOL;
	bit54_4 : BOOL;
	bit54_5 : BOOL;
	
	bit55_0 : BOOL;
	bit55_1 : BOOL;
	bit55_2 : BOOL;
	bit55_3 : BOOL;
	bit55_4 : BOOL; 
	
	bit74_0 : BOOL;
	bit74_1 : BOOL;
	bit74_2 : BOOL;
	bit74_3 : BOOL;
	bit74_4 : BOOL;
	bit74_5 : BOOL;
	
	bit75_0 : BOOL;
	bit75_1 : BOOL;
	bit75_2 : BOOL;
	bit75_3 : BOOL;
	bit75_4 : BOOL; 
	
	bit94_0 : BOOL;
	bit94_1 : BOOL;
	bit94_2 : BOOL;
	bit94_3 : BOOL;
	bit94_4 : BOOL;
	bit94_5 : BOOL;
	
	bit95_0 : BOOL;
	bit95_1 : BOOL;
	bit95_2 : BOOL;
	bit95_3 : BOOL;
	bit95_4 : BOOL; 	
	
	ID1_I0_MODE_COMMAND_0 AT %IX232.0 : BOOL :=0;
	ID1_I0_MODE_COMMAND_1 AT %IX232.1 : BOOL:=0;
	ID1_I0_READY AT %IX232.4 : BOOL;
	ID1_I0_ALARM AT %IX232.5 : BOOL;
	ID1_I0_INITIAL AT %IX232.6 : BOOL;
	ID1_I0_COMMUNICATING AT %IX232.7 : BOOL;
	ID1_I1_0 AT %IX233.0 : BOOL;
	ID1_I1_1 AT %IX233.1 : BOOL;
	ID1_I1_2 AT %IX233.2 : BOOL;
	ID1_I1_3 AT %IX233.3 : BOOL;
	ID1_I1_4 AT %IX233.4 : BOOL;
	ID1_I2_0 AT %IX234.0 : BOOL;
	ID1_I2_1 AT %IX234.1 : BOOL;
	ID1_I2_2 AT %IX234.2 : BOOL;
	ID1_I2_3 AT %IX234.3 : BOOL;
	ID1_I2_4 AT %IX234.4 : BOOL;

	ID1_I3_0 AT %IX235.0 : BOOL;
	ID1_I3_1 AT %IX235.1 : BOOL;
	
	ID1_I32_0 AT %IX264.0 : BOOL;
	ID1_I32_1 AT %IX264.1 : BOOL;
	ID1_I33_0 AT %IX265.0 : BOOL;
	ID1_I33_1 AT %IX265.1 : BOOL;
(*-----------------------------------------------------------*)

	iTest15: SINT;
	iTest16: SINT;
	
	bTest1 : BOOL;
	bTest2 : BOOL;
	bTest3 : BOOL;
	bTest4 : BOOL;
	bTest5 : BOOL;
	bTest6 : BOOL;
	bTest7 : BOOL;
	bTest8 : BOOL;
	bTest9 : BOOL;
	bTest10 : BOOL;
	bTest11 : BOOL;
	bTest12 : BOOL;
	bTest13 : BOOL;
	bTest14 : BOOL;
	
	StepData1 : BYTE;
	StepData2 : BYTE;
	StepData3 : BYTE;
	StepData4 : BYTE;
	StepData5 : BYTE;
	
	star :BOOL;
	hom : BOOL;

	reset: BOOL;
	
	ID1_ALARM AT%IX247.7 : BOOL;
	ID2_ALARM AT%IX267.7 : BOOL;
	ID3_ALARM AT%IX287.7 : BOOL;
	ID4_ALARM AT%IX307.7 : BOOL;
	ID5_ALARM AT%IX327.7 : BOOL;
	
	ID1_SVRE AT%IX247.1 : BOOL;
	ID2_SVRE AT%IX267.1 : BOOL;
	ID3_SVRE AT%IX287.1 : BOOL;
	ID4_SVRE AT%IX307.1 : BOOL;
	ID5_SVRE AT%IX327.1 : BOOL;
	
	ID1_INP AT%IX247.3 : BOOL;
	ID2_INP AT%IX267.3 : BOOL;
	ID3_INP AT%IX287.3 : BOOL;
	ID4_INP AT%IX307.3 : BOOL;
	ID5_INP AT%IX327.3 : BOOL;
	
	PROSES: STRING;
	STAGE: INT;
	
	PROCESS: INT;
	START_PROCESS: BOOL;
	STEP_DATAS: INT;
	PROCESS_DELAY: TIME :=T#300MS;
	LASER_RUNNING: BOOL :=FALSE;
	ACTIVE_STEPDATA : BYTE;
	//ACTIVE_ID: INT :=1;
	TMR1: TON;
	TMR2: TON;
	TMR3: TON;
	TMR4: TON;
	TMR5: TON;
	TMR6: TON;
	TMR10: Ton;
	TMR11: TON;
	TMR12: TON;
	TMR13: TON;
	TMR14: TON;
	TMR20: TON;
	TMR21: TON;
	TMR22: TON;
	TMR23: TON;
	TMR30: TON;
	TMR31: TON;
	TMR32: TON;
	TMR33: TON;
	TMR40: TON;
	TMR41: TON;
	TMR42: TON;
	TMR43: TON;
	TMR50: TON;
	TMR51: TON;
	TMR52: TON;
	TMR53: TON;
	
	
	TMR101: TON;
	TMR102: TON;
	TMR103: TON;
	TMR104: TON;
	TMR105: TON;
	TMR106: TON;
	ID5: INT;
	TMR7: Ton;
	TMR_RES_CARTSN: TOF;
	TMR_ACTIVATE_RESET: TON;
END_VAR


PROCESS_DELAY:= T#400MS;
IF 	SORTER_VAR.ACTIVE_ID >=0 THEN
STEP_DATA_1:=STEP_DATA_1+1;

IF STEP_DATA_2>=5 THEN
	STEP_DATA_2:=STEP_DATA_2+1;
END_IF

STEP_DATA_3:=STEP_DATA_3+1;	
END_IF


IF NOT SORTER_VAR.LASER_HOME THEN //LASER_running THEN
	IF  ID1_SVRE AND ID2_SVRE  AND  ID3_SVRE AND  ID4_SVRE AND  ID5_SVRE THEN
		TMR1(IN:=TRUE,PT:=T#0.5S);
		TMR4(IN:=TRUE,PT:=T#3S);
		TMR5(IN:=TRUE,PT:=T#3.5S);
		TMR6(IN:=TRUE,PT:=T#25S);
		IF ID1_SVRE THEN
			ID1_SETUP :=TMR5.Q;
		ELSE
			ID1_SVON :=TRUE;	
		END_IF

		IF ID2_SVRE THEN
			ID2_SETUP :=TMR1.Q;
		ELSE
			ID2_SVON :=TRUE;	
		END_IF
	
		IF ID3_SVRE THEN
		ID3_SETUP :=TMR4.Q;
		ELSE
			ID3_SVON :=TRUE;	
		END_IF
		CASE SORTER_VAR.I_CURRENT_TRANSACTION.TRANSPORT_INDEX OF
		1:
			TMR2(IN:=TRUE,PT:=T#1S);
			IF ID4_SVRE THEN
				ID4_SETUP :=TMR2.Q;
			ELSE
				ID4_SVON :=TRUE;	
			END_IF
		2:
			TMR3(IN:=TRUE,PT:=T#1.5S);
			IF ID5_SVRE THEN
				ID5_SETUP :=TMR3.Q;
			ELSE
				ID5_SVON :=TRUE;	
			END_IF
		END_CASE

	//IF TMR6.Q THEN
	IF ID1_INP AND ID2_INP AND ID3_INP AND (ID4_INP OR ID5_INP) THEN
		ID1_SETUP :=FALSE;
		ID2_SETUP :=FALSE;
		ID3_SETUP :=FALSE;
		ID4_SETUP :=FALSE;
		ID5_SETUP :=FALSE;
	
		TMR1(IN:=FALSE);
		TMR2(IN:=FALSE);
		TMR3(IN:=FALSE);
		TMR4(IN:=FALSE);
		TMR5(IN:=FALSE);
	//ACTIVE_ID:=1;
	//LASER_RUNNING:=TRUE;
		SORTER_VAR.LASER_HOME:=TRUE;
	END_IF
	
	ELSE
				
	ID1_SVON :=TRUE;
	ID2_SVON :=TRUE;
	ID3_SVON :=TRUE;
	ID4_SVON :=TRUE;
	ID5_SVON :=TRUE;

	END_IF
ELSE
	TMR6(IN:=FALSE);

	CASE SORTER_VAR.ACTIVE_ID OF
	0:
		SORTER_VAR.I_CASE:=SORTER_VAR.I_CASE+1;
		//SORTER_VAR.I_LASER_RUNNING:=FALSE;
		SORTER_VAR.ACTIVE_ID:=6;
		
	1:
		IF STEP_DATA_1 = 0 THEN
			SORTER_VAR.ACTIVE_ID:=2;
		ELSE
			IF ID1_ALARM THEN
				Reset := TRUE;
				TMR10(IN:=TRUE,PT:= PROCESS_DELAY);
				IF TMR10.Q THEN
					Reset := FALSE;
				END_IF
			ELSE
				ID1_StepData :=STEP_DATA_1;
				ID1_Drive := FALSE;
				TMR11(IN:=TRUE,PT:= PROCESS_DELAY);
				IF TMR11.Q THEN
					ID1_Drive := TRUE;
					TMR12(IN:=TMR11.Q,PT:= PROCESS_DELAY);
					IF TMR12.Q THEN
						ID1_Drive := FALSE;
						SORTER_VAR.ACTIVE_ID:=2;
						TMR10(IN:=FALSE);
						TMR11(IN:=FALSE);
						TMR12(IN:=FALSE);
						SORTER_VAR.LASER_HOME:=TRUE;
					END_IF
				END_IF
			END_IF
		END_IF
	//	SORTER_VAR.I_CASE:=SORTER_VAR.I_CASE+1;
		//SORTER_VAR.I_LASER_RUNNING:=FALSE;
	2:
		IF STEP_DATA_2 = 0 THEN
			SORTER_VAR.ACTIVE_ID:=3;
		ELSE
			
			IF ID2_ALARM THEN
				Reset := TRUE;
				TMR20(IN:=TRUE,PT:= PROCESS_DELAY);
				IF TMR20.Q THEN
					Reset := FALSE;
				END_IF
			ELSE
			ID2_StepData :=STEP_DATA_2;
			TMR21(IN:=TRUE,PT:= PROCESS_DELAY);
			IF TMR21.Q THEN
				ID2_Drive := TRUE;
				TMR22(IN:=TMR21.Q,PT:= PROCESS_DELAY);
				IF TMR22.Q THEN
		
					ID2_Drive := FALSE;
					SORTER_VAR.ACTIVE_ID:=3;
					TMR20(IN:=FALSE);
					TMR21(IN:=FALSE);
					TMR22(IN:=FALSE);
				END_IF
			END_IF
			END_IF
		END_IF
	3:
		IF STEP_DATA_3 = 0 THEN
			SORTER_VAR.ACTIVE_ID:=4;
		ELSE
			
		IF ID3_ALARM THEN
			Reset := TRUE;
			TMR30(IN:=START_PROCESS,PT:= PROCESS_DELAY);
			IF TMR30.Q THEN
				Reset := FALSE;
			END_IF
		ELSE
		
		ID3_StepData :=STEP_DATA_3;
		TMR31(IN:=TRUE,PT:= PROCESS_DELAY);
		IF TMR31.Q THEN
			ID3_DRIVE := TRUE;	
			TMR32(IN:=TMR31.Q,PT:= PROCESS_DELAY);
			
			IF TMR32.Q THEN
				ID3_Drive := FALSE;
				SORTER_VAR.ACTIVE_ID:=4;
				TMR30(IN:=FALSE);
				TMR31(IN:=FALSE);
				TMR32(IN:=FALSE);
			END_IF
		END_IF
		END_IF
	END_IF
4:
		IF STEP_DATA_4 = 0 THEN
			SORTER_VAR.ACTIVE_ID:=5;
		ELSE
			IF ID4_ALARM THEN
				Reset := TRUE;
				TMR40(IN:=TRUE,PT:= PROCESS_DELAY);
				IF TMR40.Q THEN
					Reset := FALSE;
				END_IF
			ELSE
			
			ID4_StepData :=STEP_DATA_4;
			TMR41(IN:=TRUE,PT:= PROCESS_DELAY);
			IF TMR41.Q THEN
				ID4_Drive := TRUE;
				TMR42(IN:=TMR41.Q,PT:= PROCESS_DELAY);
				
				IF TMR42.Q THEN
					ID4_Drive := FALSE;
					SORTER_VAR.ACTIVE_ID:=5;
					TMR40(IN:=FALSE);
					TMR41(IN:=FALSE);
					TMR42(IN:=FALSE);
				END_IF
			END_IF
			END_IF
		END_IF
	5:
		IF STEP_DATA_5 = 0 THEN
			SORTER_VAR.ACTIVE_ID:=0;
		ELSE
			
			IF ID5_ALARM THEN
				Reset := TRUE;
				TMR50(IN:=TRUE,PT:= PROCESS_DELAY);
				IF TMR50.Q THEN
					Reset := FALSE;
				END_IF
			ELSE
			
			ID5_StepData :=STEP_DATA_5;
			TMR51(IN:=TRUE,PT:= PROCESS_DELAY);
			IF TMR51.Q THEN
				ID5_Drive := TRUE;	
				TMR52(IN:=TMR51.Q,PT:= PROCESS_DELAY);
				IF TMR52.Q THEN
					ID5_Drive := FALSE;
					SORTER_VAR.ACTIVE_ID:=0;
					TMR50(IN:=FALSE);
					TMR51(IN:=FALSE);
					TMR52(IN:=FALSE);
			
				END_IF
			END_IF
			END_IF
		END_IF
		
END_CASE 

	//START_PROCESS := FALSE;
END_IF
TMR7(IN:=reset,PT:= T#1S);
IF  tmr7.Q THEN
	reset:=FALSE;
END_IF
IF ID1_ALARM OR ID2_ALARM OR ID3_ALARM OR ID4_ALARM OR ID5_ALARM THEN
			reset:=TRUE;
			ELSE
				reset:=FALSE;
			END_IF
IF reset THEN
	ID1_Reset := TRUE;
	ID2_Reset := TRUE;
	ID3_Reset := TRUE;
	ID4_Reset := TRUE;
	ID5_Reset := TRUE;
	TMR_ACTIVATE_RESET(IN:=TRUE,PT:=T#10S);
	IF TMR_ACTIVATE_RESET.Q THEN
		TMR_RES_CARTSN(IN:=TRUE,PT:=T#0.5S);
	END_IF
	
ELSE
	TMR_ACTIVATE_RESET(IN:=FALSE);
	TMR_RES_CARTSN(IN:=FALSE);
	ID1_Reset := FALSE;
	ID2_Reset := FALSE;
	ID3_Reset := FALSE;
	ID4_Reset := FALSE;
	ID5_Reset := FALSE;
END_IF
SORTER_VAR.O_RESET_CARTESSIAN := TMR_RES_CARTSN.Q;

END_PROGRAM

// ---- POUs/LASER/RETURN_LASER.TcPOU
PROGRAM RETURN_LASER
VAR_INPUT

END_VAR

VAR
	TMR_DELAY: TON;
	TMR_DELAY1: TON;
	TMR_DELAY2: TON;
END_VAR

CASE SORTER_VAR.I_CASE OF
0: //standby near lotbox
	IF SORTER_VAR.ACTIVE_ID=6 THEN
		SORTER_VAR.ACTIVE_ID:=1;
	END_IF

	CASE SORTER_VAR.I_CURRENT_TRANSACTION.TRANSPORT_INDEX OF
		2 : 
			SORTER_VAR.O_STOPPER_TRANSFER_B:=FALSE;			
			LASER_MOVE(STEP_DATA_1:=0,//3,
				STEP_DATA_2:=1,
				STEP_DATA_3:=12,
				STEP_DATA_4:=0,
				STEP_DATA_5:=1);
		1 : 
			SORTER_VAR.O_STOPPER_TRANSFER_A:=FALSE;
			LASER_MOVE(STEP_DATA_1:=0,//3,
				STEP_DATA_2:=1,
				STEP_DATA_3:=12,
				STEP_DATA_4:=1,
				STEP_DATA_5:=0);
	END_CASE			
	SORTER_VAR.O_VACUUM_On:=FALSE;
	SORTER_VAR.O_VACUUM_OFF:=FALSE;	
	TMR_DELAY(IN:=FALSE);

1://ready for picking up
	IF SORTER_VAR.ACTIVE_ID=6 THEN
		SORTER_VAR.ACTIVE_ID:=1;
	END_IF

		CASE SORTER_VAR.I_CURRENT_TRANSACTION.TRANSPORT_INDEX OF
		1:
			SORTER_VAR.I_RETURN_DONE_A:=FALSE;
		
		2:
			SORTER_VAR.I_RETURN_DONE_B:=FALSE;
	END_CASE
	LASER_MOVE(STEP_DATA_1:=0,
				STEP_DATA_2:=1,
				STEP_DATA_3:=11,
				STEP_DATA_4:=0,
				STEP_DATA_5:=0);	
			
2://ready for picking up
	IF SORTER_VAR.ACTIVE_ID=6 THEN
		SORTER_VAR.ACTIVE_ID:=1;
	END_IF
	TMR_DELAY(IN:=TRUE,PT:=T#1S);
	IF TMR_DELAY.Q THEN
	CASE SORTER_VAR.I_CURRENT_TRANSACTION.TRANSPORT_INDEX OF
	1:		
		//IF SORTER_VAR.I_LASER_TRANSFER_AT_BACK_A THEN
		LASER_MOVE(STEP_DATA_1:=SORTER_VAR.I_CURRENT_TRANSACTION.TRANSPORT_INDEX+5,
				STEP_DATA_2:=1,
				STEP_DATA_3:=11,
				STEP_DATA_4:=0,
				STEP_DATA_5:=0);
		//END_IF
	2:
		//IF SORTER_VAR.I_LASER_TRANSFER_AT_BACK_B THEN
		LASER_MOVE(STEP_DATA_1:=SORTER_VAR.I_CURRENT_TRANSACTION.TRANSPORT_INDEX+5,
				STEP_DATA_2:=1,
				STEP_DATA_3:=11,
				STEP_DATA_4:=0,
				STEP_DATA_5:=0);
	//END_IF
	END_CASE
	END_IF
		
3://VACUUM AND TAKEUP
	IF SORTER_VAR.ACTIVE_ID=6 THEN
		SORTER_VAR.ACTIVE_ID:=1;
	END_IF

	LASER_MOVE(STEP_DATA_1:=SORTER_VAR.I_CURRENT_TRANSACTION.TRANSPORT_INDEX+5,
				STEP_DATA_2:=5,
				STEP_DATA_3:=11,
				STEP_DATA_4:=0,
				STEP_DATA_5:=0);
	SORTER_VAR.O_VACUUM_On:=TRUE;
	SORTER_VAR.O_VACUUM_OFF:=FALSE;
	
4://MOVE BACK 10MM
	IF SORTER_VAR.ACTIVE_ID=6 THEN
		SORTER_VAR.ACTIVE_ID:=1;
	END_IF
	
	LASER_MOVE(STEP_DATA_1:=SORTER_VAR.I_CURRENT_TRANSACTION.TRANSPORT_INDEX+5,
				STEP_DATA_2:=1,
				STEP_DATA_3:=12,
				STEP_DATA_4:=0,
				STEP_DATA_5:=0);

5://MOVE UP 16MM
	IF SORTER_VAR.ACTIVE_ID=6 THEN
		SORTER_VAR.ACTIVE_ID:=1;
	END_IF
	LASER_MOVE(STEP_DATA_1:=SORTER_VAR.I_CURRENT_TRANSACTION.TRANSPORT_INDEX+5,
				STEP_DATA_2:=1,
				STEP_DATA_3:=SORTER_VAR.I_CURRENT_TRANSACTION.JIG_INDEX_RETURN,
				STEP_DATA_4:=0,
				STEP_DATA_5:=0);
	(*
	IF NOT SORTER_VAR.I_VACUUM_On THEN
		LASER_MOVE(STEP_DATA_1:=SORTER_VAR.I_CURRENT_TRANSACTION.TRANSPORT_INDEX+5,
				STEP_DATA_2:=2,
				STEP_DATA_3:=12,
				STEP_DATA_4:=0,
				STEP_DATA_5:=0);
	ELSE
		SORTER_VAR.O_VACUUM_On:=TRUE;
		SORTER_VAR.O_VACUUM_OFF:=FALSE;
	END_IF
	*)
				
6://WAIT THEN MOVE TO NEAR BOX
	IF SORTER_VAR.ACTIVE_ID=6 THEN
		SORTER_VAR.ACTIVE_ID:=1;
	END_IF
	TMR_DELAY1(IN:=TRUE,PT:=T#3S);
	IF TMR_DELAY1.Q THEN
		LASER_MOVE(STEP_DATA_1:=SORTER_VAR.I_CURRENT_TRANSACTION.STATION_NUMBER_RETURN,
				STEP_DATA_2:=2,
				STEP_DATA_3:=14,
				STEP_DATA_4:=0,
				STEP_DATA_5:=0);
	END_IF
	
				
7://vacuum position 
	IF SORTER_VAR.ACTIVE_ID=6 THEN
		SORTER_VAR.ACTIVE_ID:=1;
	END_IF
	SORTER_VAR.I_CASE:=SORTER_VAR.I_CASE+1;
	(*
	TMR_DELAY(IN:=TRUE,PT:=T#1S);
	IF TMR_DELAY.Q THEN
			LASER_MOVE(STEP_DATA_1:=SORTER_VAR.I_CURRENT_TRANSACTION.STATION_NUMBER_RETURN,
				STEP_DATA_2:=2,
				STEP_DATA_3:=14,
				STEP_DATA_4:=0,
				STEP_DATA_5:=0);
	END_IF
		*)		
8://INSERT INTO LOTBOX
	IF SORTER_VAR.ACTIVE_ID=6 THEN
		SORTER_VAR.ACTIVE_ID:=1;
	END_IF
	TMR_DELAY(IN:=FALSE);
	LASER_MOVE(STEP_DATA_1:=SORTER_VAR.I_CURRENT_TRANSACTION.STATION_NUMBER_RETURN,
				STEP_DATA_2:=3,
				STEP_DATA_3:=16,
				STEP_DATA_4:=0,
				STEP_DATA_5:=0);
				
9://MOVE BACK
	IF SORTER_VAR.ACTIVE_ID=6 THEN
		SORTER_VAR.ACTIVE_ID:=1;
	END_IF
	TMR_DELAY2 (IN:=TRUE,PT:=T#2S);
	IF TMR_DELAY2.Q THEN
		LASER_MOVE(STEP_DATA_1:=SORTER_VAR.I_CURRENT_TRANSACTION.STATION_NUMBER_RETURN,
				STEP_DATA_2:=3,
				STEP_DATA_3:=SORTER_VAR.I_CURRENT_TRANSACTION.JIG_INDEX_RETURN,
				STEP_DATA_4:=0,
				STEP_DATA_5:=0);
	END_IF
	SORTER_VAR.O_VACUUM_On:=FALSE;
	SORTER_VAR.O_VACUUM_OFF:=TRUE;
10: //standby near lotbox
	
	IF SORTER_VAR.ACTIVE_ID=6 THEN
		SORTER_VAR.ACTIVE_ID:=1;
	END_IF
LASER_MOVE(STEP_DATA_1:=SORTER_VAR.I_CURRENT_TRANSACTION.STATION_NUMBER_RETURN,
				STEP_DATA_2:=1,
				STEP_DATA_3:=SORTER_VAR.I_CURRENT_TRANSACTION.JIG_INDEX_RETURN,
				STEP_DATA_4:=0,
				STEP_DATA_5:=0);
	(*
	IF SORTER_VAR.I_VACUUM_ON THEN
		LASER_MOVE(STEP_DATA_1:=SORTER_VAR.I_CURRENT_TRANSACTION.STATION_NUMBER_RETURN,
				STEP_DATA_2:=4,
				STEP_DATA_3:=SORTER_VAR.I_CURRENT_TRANSACTION.JIG_INDEX_RETURN,
				STEP_DATA_4:=0,
				STEP_DATA_5:=0);
	ELSE
		SORTER_VAR.O_VACUUM_ON:=FALSE;
		SORTER_VAR.O_VACUUM_OFF:=TRUE;			
	END_IF
	*)
				
11://vacuum position 
	IF SORTER_VAR.ACTIVE_ID=6 THEN
		SORTER_VAR.ACTIVE_ID:=1;
	END_IF
	LASER_MOVE(STEP_DATA_1:=0,
				STEP_DATA_2:=1,
				STEP_DATA_3:=4,
				STEP_DATA_4:=0,
				STEP_DATA_5:=0);
	IF SORTER_VAR.ACTIVE_ID=3 THEN
		SORTER_VAR.O_VACUUM_ON:=FALSE;
		SORTER_VAR.O_VACUUM_OFF:=FALSE;	
	END_IF
	
			
		
100:
	
	SORTER_VAR.O_VACUUM_On:=FALSE;
	SORTER_VAR.O_VACUUM_OFF:=FALSE;
END_CASE 
IF SORTER_VAR.I_CASE=12 THEN
			CASE SORTER_VAR.I_CURRENT_TRANSACTION.TRANSPORT_INDEX OF
		1:
			SORTER_VAR.I_RETURN_DONE_A:=TRUE;
		
		2:
			SORTER_VAR.I_RETURN_DONE_B:=TRUE;
	END_CASE
	IF SORTER_VAR.I_RETURN_DONE_A OR SORTER_VAR.I_RETURN_DONE_B THEN
		FLAG_VAR.ALLOW_EXECUTE_RETURN_LASER:=FALSE;
		TMR_DELAY(IN:=FALSE);
		TMR_DELAY1(IN:=FALSE);
		TMR_DELAY2(IN:=FALSE);
		
		SORTER_VAR.I_CASE:=100;
	END_IF
END_IF

END_PROGRAM

// ---- POUs/LASER/LOAD_NG.TcPOU
PROGRAM LOAD_NG
VAR
	DELAY: TON;
END_VAR

IF NOT SORTER_VAR.I_NG_TRANSFER_AT_BACK THEN
	SORTER_VAR.O_NG_DATA_OUTPUT2:=TRUE;
ELSE
	SORTER_VAR.O_NG_DATA_OUTPUT2:=FALSE;
END_IF

END_PROGRAM

// ---- POUs/LASER/RETURN_NG.TcPOU
PROGRAM RETURN_NG
VAR
	DELAY: TON;
END_VAR

IF NOT SORTER_VAR.I_NG_TRANSFER_AT_FRONT THEN
	SORTER_VAR.O_NG_DATA_OUTPUT1:=TRUE;
ELSE
	SORTER_VAR.O_NG_DATA_OUTPUT1:=FALSE;
END_IF

END_PROGRAM

// ---- POUs/EXECUTE_FUNCTION.TcPOU
FUNCTION EXECUTE_FUNCTION : BOOL
VAR_INPUT
	FUNCT_NAME :STRING [255];
END_VAR
VAR
END_VAR

IF FUNCT_NAME = 'LOAD_FUKUDA' THEN
	//LOAD_FUKUDA(INPUT_VAR.I_CURRENT_TRANSACTION.STATION_NUMBER_LOAD,INPUT_VAR.I_CURRENT_TRANSACTION.JIG_INDEX_LOAD,INPUT_VAR.I_CURRENT_TRANSACTION.TRANSPORT_INDEX);
	INPUT_VAR.I_FUNC_CALLED:=TRUE;
	LOAD_FUKUDA();
END_IF
//INPUT_VAR.I_FUNCTION_NAME:='';

END_FUNCTION

// ---- POUs/FUKUDA/FUKUDA_MOVE_1.TcPOU
PROGRAM FUKUDA_MOVE_1
//FUNCTION FUKUDA_MOVE : BOOL
VAR_INPUT
	STEP_DATA_1: BYTE;
	STEP_DATA_2: BYTE;
	STEP_DATA_3: BYTE;
	STEP_DATA_4: BYTE;
	STEP_DATA_5: BYTE;
	FUKUDA_HOME: INT;
END_VAR

VAR
	
	(*
	DataWordInput1 AT %IB100 : ARRAY [0..15] OF WORD; 
	DataWordInput2 AT %IB132 : ARRAY [16..31] OF WORD; 
	DataWordInput3 AT %IB164 : ARRAY [32..47] OF WORD; 
	DataWordInput4 AT %IB196 : ARRAY [48..56] OF WORD; 
	DataWordOutput1 AT %QB100 : ARRAY [0..15] OF WORD; 
	DataWordOutput2 AT %QB132 : ARRAY [16..31] OF WORD; 
	DataWordOutput3 AT %QB164 : ARRAY [32..47] OF WORD; 
	DataWordOutput4 AT %QB196 : ARRAY [48..56] OF WORD; 
	*)
	Gateway_Q0_MODE_COMMAND_0 AT %QX100.0 : BOOL ;
	Gateway_Q0_MODE_COMMAND_1 AT %QX100.1 : BOOL ;
	Gateway_Q0_RESET AT %QX100.4 : BOOL;
	Gateway_Q0_RESTART AT %QX100.5 : BOOL;
	Gateway_Q0_STOP AT %QX100.7 : BOOL;
	Gateway_Q1_0 AT %QX101.0 : BOOL;
	Gateway_Q1_1 AT %QX101.1 : BOOL;
	Gateway_Q1_2 AT %QX101.2 : BOOL;
	Gateway_Q1_3 AT %QX101.3 : BOOL;
	Gateway_Q1_4 AT %QX101.4 : BOOL;
	Gateway_Gateway_Unit_2_Status AT %QB102 : BYTE;
	Gateway_Q3_0 AT %QX103.0 : BOOL;
	Gateway_Q3_1 AT %QX103.1 : BOOL;
	Gateway_Q3_2 AT %QX103.2 : BOOL;
	Gateway_Q3_3 AT %QX103.3 : BOOL;	
	

	ID1_StepData AT %QB114 : BYTE;
	ID1_Hold AT %QX115.0 : BOOL;
	ID1_SVON AT %QX115.1 : BOOL;
	ID1_Drive AT %QX115.2 : BOOL;
	ID1_Reset AT %QX115.3 : BOOL;
	ID1_Setup AT %QX115.4 : BOOL;
	

	ID2_StepData AT %QB134 : BYTE;
	ID2_Hold AT %QX135.0 : BOOL;
	ID2_SVON AT %QX135.1 : BOOL;
	ID2_Drive AT %QX135.2 : BOOL;
	ID2_Reset AT %QX135.3 : BOOL;
	ID2_Setup AT %QX135.4 : BOOL;


	ID3_StepData AT %QB154 : BYTE;
	ID3_Hold AT %QX155.0 : BOOL;
	ID3_SVON AT %QX155.1 : BOOL;
	ID3_Drive AT %QX155.2 : BOOL;
	ID3_Reset AT %QX155.3 : BOOL;
	ID3_Setup AT %QX155.4 : BOOL;
	
	
	ID4_StepData AT %QB174 : BYTE;
	ID4_Hold AT %QX175.0 : BOOL;
	ID4_SVON AT %QX175.1 : BOOL;
	ID4_Drive AT %QX175.2 : BOOL;
	ID4_Reset AT %QX175.3 : BOOL;
	ID4_Setup AT %QX175.4 : BOOL;
	

	ID5_StepData AT %QB194 : BYTE;
	ID5_Hold AT %QX195.0 : BOOL;
	ID5_SVON AT %QX195.1 : BOOL;
	ID5_Drive AT %QX195.2 : BOOL;
	ID5_Reset AT %QX195.3 : BOOL;
	ID5_Setup AT %QX195.4 : BOOL;
	
	byte0 : BYTE;
	byte1 : BYTE;
	byte2 : BYTE;
	byte3 : BYTE;
	
	bit14_0 : BOOL;
	bit14_1 : BOOL;
	bit14_2 : BOOL;
	bit14_3 : BOOL;
	bit14_4 : BOOL;
	bit14_5 : BOOL;
	
	bit15_0 : BOOL;
	bit15_1 : BOOL;
	bit15_2 : BOOL;
	bit15_3 : BOOL;
	bit15_4 : BOOL; 
	
	bit34_0 : BOOL;
	bit34_1 : BOOL;
	bit34_2 : BOOL;
	bit34_3 : BOOL;
	bit34_4 : BOOL;
	bit34_5 : BOOL;
	
	bit35_0 : BOOL;
	bit35_1 : BOOL;
	bit35_2 : BOOL;
	bit35_3 : BOOL;
	bit35_4 : BOOL; 
	
	bit54_0 : BOOL;
	bit54_1 : BOOL;
	bit54_2 : BOOL;
	bit54_3 : BOOL;
	bit54_4 : BOOL;
	bit54_5 : BOOL;
	
	bit55_0 : BOOL;
	bit55_1 : BOOL;
	bit55_2 : BOOL;
	bit55_3 : BOOL;
	bit55_4 : BOOL; 
	
	bit74_0 : BOOL;
	bit74_1 : BOOL;
	bit74_2 : BOOL;
	bit74_3 : BOOL;
	bit74_4 : BOOL;
	bit74_5 : BOOL;
	
	bit75_0 : BOOL;
	bit75_1 : BOOL;
	bit75_2 : BOOL;
	bit75_3 : BOOL;
	bit75_4 : BOOL; 
	
	bit94_0 : BOOL;
	bit94_1 : BOOL;
	bit94_2 : BOOL;
	bit94_3 : BOOL;
	bit94_4 : BOOL;
	bit94_5 : BOOL;
	
	bit95_0 : BOOL;
	bit95_1 : BOOL;
	bit95_2 : BOOL;
	bit95_3 : BOOL;
	bit95_4 : BOOL; 	
	
	ID1_I0_MODE_COMMAND_0 AT %IX100.0 : BOOL :=0;
	ID1_I0_MODE_COMMAND_1 AT %IX100.1 : BOOL:=0;
	ID1_I0_READY AT %IX100.4 : BOOL;
	ID1_I0_ALARM AT %IX100.5 : BOOL;
	ID1_I0_INITIAL AT %IX100.6 : BOOL;
	ID1_I0_COMMUNICATING AT %IX100.7 : BOOL;
	ID1_I1_0 AT %IX101.0 : BOOL;
	ID1_I1_1 AT %IX101.1 : BOOL;
	ID1_I1_2 AT %IX101.2 : BOOL;
	ID1_I1_3 AT %IX101.3 : BOOL;
	ID1_I1_4 AT %IX101.4 : BOOL;
	ID1_I2_0 AT %IX102.0 : BOOL;
	ID1_I2_1 AT %IX102.1 : BOOL;
	ID1_I2_2 AT %IX102.2 : BOOL;
	ID1_I2_3 AT %IX102.3 : BOOL;
	ID1_I2_4 AT %IX102.4 : BOOL;

	ID1_I3_0 AT %IX103.0 : BOOL;
	ID1_I3_1 AT %IX103.1 : BOOL;
	
	ID1_I32_0 AT %IX132.0 : BOOL;
	ID1_I32_1 AT %IX132.1 : BOOL;
	ID1_I33_0 AT %IX133.0 : BOOL;
	ID1_I33_1 AT %IX133.1 : BOOL;
(*-----------------------------------------------------------*)

	iTest15: SINT;
	iTest16: SINT;
	
	bTest1 : BOOL;
	bTest2 : BOOL;
	bTest3 : BOOL;
	bTest4 : BOOL;
	bTest5 : BOOL;
	bTest6 : BOOL;
	bTest7 : BOOL;
	bTest8 : BOOL;
	bTest9 : BOOL;
	bTest10 : BOOL;
	bTest11 : BOOL;
	bTest12 : BOOL;
	bTest13 : BOOL;
	bTest14 : BOOL;
	
	StepData1 : BYTE;
	StepData2 : BYTE;
	StepData3 : BYTE;
	StepData4 : BYTE;
	StepData5 : BYTE;
	
	star :BOOL;
	hom : BOOL;

	reset: BOOL;
	
	ID1_ALARM AT%IX115.7 : BOOL;
	ID2_ALARM AT%IX135.7 : BOOL;
	ID3_ALARM AT%IX155.7 : BOOL;
	ID4_ALARM AT%IX175.7 : BOOL;
	ID5_ALARM AT%IX195.7 : BOOL;
	
	ID1_SVRE AT%IX115.1 : BOOL;
	ID2_SVRE AT%IX135.1 : BOOL;
	ID3_SVRE AT%IX155.1 : BOOL;
	ID4_SVRE AT%IX175.1 : BOOL;
	ID5_SVRE AT%IX195.1 : BOOL;
	
	ID1_INP AT%IX115.3 : BOOL;
	ID2_INP AT%IX135.3 : BOOL;
	ID3_INP AT%IX155.3 : BOOL;
	ID4_INP AT%IX175.3 : BOOL;
	ID5_INP AT%IX195.3 : BOOL;
	
	PROSES: STRING;
	STAGE: INT;
	
	PROCESS: INT;
	START_PROCESS: BOOL;
	STEP_DATAS: INT;
	PROCESS_DELAY: TIME :=T#300MS;
	FUKUDA_RUNNING: BOOL :=FALSE;
	ACTIVE_STEPDATA : BYTE;
	//ACTIVE_ID: INT :=1;
	TMR1: TON;
	TMR2: TON;
	TMR3: TON;
	TMR4: TON;
	TMR5: TON;
	TMR6: TON;
	TMR10: Ton;
	TMR11: TON;
	TMR12: TON;
	TMR13: TON;
	TMR14: TON;
	TMR20: TON;
	TMR21: TON;
	TMR22: TON;
	TMR23: TON;
	TMR30: TON;
	TMR31: TON;
	TMR32: TON;
	TMR33: TON;
	TMR40: TON;
	TMR41: TON;
	TMR42: TON;
	TMR43: TON;
	TMR50: TON;
	TMR51: TON;
	TMR52: TON;
	TMR53: TON;
	
	
	TMR101: TON;
	TMR102: TON;
	TMR103: TON;
	TMR104: TON;
	TMR105: TON;
	TMR106: TON;
	ID5: INT;
	TMR7: Ton;
END_VAR


PROCESS_DELAY:= T#400MS;
IF 	INPUT_VAR.ACTIVE_ID >=0 THEN
STEP_DATA_1:=STEP_DATA_1+1;

IF STEP_DATA_2>=5 THEN
	STEP_DATA_2:=STEP_DATA_2+1;
END_IF

STEP_DATA_3:=STEP_DATA_3+1;	
END_IF


IF NOT INPUT_VAR.FUKUDA_HOME THEN //fukuda_running THEN
	IF  ID1_SVRE AND ID2_SVRE  AND  ID3_SVRE AND  ID4_SVRE AND  ID5_SVRE THEN
		(*
IF ID1_ALARM THEN
		RESET:=TRUE;
		ELSE
		RESET:=FALSE;	
	END_IF
	*)

	TMR1(IN:=TRUE,PT:=T#0.5S);
	TMR4(IN:=TRUE,PT:=T#3S);
	TMR5(IN:=TRUE,PT:=T#3.5S);
	TMR6(IN:=TRUE,PT:=T#25S);
	//RESET := FALSE;	
	
	IF ID1_SVRE THEN
		ID1_SETUP :=TMR4.Q;
	ELSE
		ID1_SVON :=TRUE;	
	END_IF

	IF ID2_SVRE THEN
		ID2_SETUP :=TMR1.Q;
	ELSE
		ID2_SVON :=TRUE;	
	END_IF
	
	IF ID3_SVRE THEN
	ID3_SETUP :=TMR5.Q;
	ELSE
		ID3_SVON :=TRUE;	
	END_IF
		CASE INPUT_VAR.I_CURRENT_TRANSACTION.TRANSPORT_INDEX OF
		1:
			TMR2(IN:=TRUE,PT:=T#1S);
			IF ID4_SVRE THEN
				ID4_SETUP :=TMR2.Q;
			ELSE
				ID4_SVON :=TRUE;	
			END_IF
		2:
			TMR3(IN:=TRUE,PT:=T#1.5S);
			IF ID5_SVRE THEN
				ID5_SETUP :=TMR3.Q;
			ELSE
				ID5_SVON :=TRUE;	
			END_IF
		END_CASE

	//IF TMR6.Q THEN
	IF ID1_INP AND ID2_INP AND ID3_INP AND (ID4_INP OR ID5_INP) THEN
		ID1_SETUP :=FALSE;
		ID2_SETUP :=FALSE;
		ID3_SETUP :=FALSE;
		ID4_SETUP :=FALSE;
		ID5_SETUP :=FALSE;
	
		TMR1(IN:=FALSE);
		TMR2(IN:=FALSE);
		TMR3(IN:=FALSE);
		TMR4(IN:=FALSE);
		TMR5(IN:=FALSE);
	//ACTIVE_ID:=1;
	//FUKUDA_RUNNING:=TRUE;
		INPUT_VAR.FUKUDA_HOME:=TRUE;
	END_IF
	
	ELSE
				
	ID1_SVON :=TRUE;
	ID2_SVON :=TRUE;
	ID3_SVON :=TRUE;
	ID4_SVON :=TRUE;
	ID5_SVON :=TRUE;

	END_IF
ELSE
	TMR6(IN:=FALSE);

	CASE INPUT_VAR.ACTIVE_ID OF
	0:
		INPUT_VAR.I_CASE:=INPUT_VAR.I_CASE+1;
		//INPUT_VAR.I_FUKUDA_RUNNING:=FALSE;
		INPUT_VAR.ACTIVE_ID:=6;
		
	1:
		IF STEP_DATA_1 = 0 THEN
			INPUT_VAR.ACTIVE_ID:=2;
		ELSE
			IF ID1_ALARM THEN
				Reset := TRUE;
				TMR10(IN:=TRUE,PT:= PROCESS_DELAY);
				IF TMR10.Q THEN
					Reset := FALSE;
				END_IF
			END_IF
			ID1_StepData :=STEP_DATA_1;
			TMR11(IN:=TRUE,PT:= PROCESS_DELAY);
			IF TMR11.Q THEN
				ID1_Drive := TRUE;
				TMR12(IN:=TMR11.Q,PT:= PROCESS_DELAY);
				IF TMR12.Q THEN
				
					ID1_Drive := FALSE;
					INPUT_VAR.ACTIVE_ID:=2;
					TMR10(IN:=FALSE);
					TMR11(IN:=FALSE);
					TMR12(IN:=FALSE);
					INPUT_VAR.FUKUDA_HOME:=TRUE;
				END_IF
			END_IF
		END_IF
	//	INPUT_VAR.I_CASE:=INPUT_VAR.I_CASE+1;
		//INPUT_VAR.I_FUKUDA_RUNNING:=FALSE;
	2:
		IF STEP_DATA_2 = 0 THEN
			INPUT_VAR.ACTIVE_ID:=3;
		ELSE
			
			IF ID2_ALARM THEN
				Reset := TRUE;
				TMR20(IN:=TRUE,PT:= PROCESS_DELAY);
				IF TMR20.Q THEN
								Reset := FALSE;
				END_IF
			END_IF
			
			ID2_StepData :=STEP_DATA_2;
			TMR21(IN:=TRUE,PT:= PROCESS_DELAY);
			IF TMR21.Q THEN
				ID2_Drive := TRUE;
				TMR22(IN:=TMR21.Q,PT:= PROCESS_DELAY);
				IF TMR22.Q THEN
		
					ID2_Drive := FALSE;
					INPUT_VAR.ACTIVE_ID:=3;
					TMR20(IN:=FALSE);
					TMR21(IN:=FALSE);
					TMR22(IN:=FALSE);
				END_IF
			END_IF
		END_IF
	3:
		IF STEP_DATA_3 = 0 THEN
			INPUT_VAR.ACTIVE_ID:=4;
		ELSE
			(*
		IF ID3_ALARM THEN
			Reset := TRUE;
			TMR30(IN:=START_PROCESS,PT:= PROCESS_DELAY);
			IF TMR30.Q THEN
				Reset := FALSE;
			END_IF
		END_IF
		*)
		ID3_StepData :=STEP_DATA_3;
		TMR31(IN:=TRUE,PT:= PROCESS_DELAY);
		IF TMR31.Q THEN
			ID3_DRIVE := TRUE;	
			TMR32(IN:=TMR31.Q,PT:= PROCESS_DELAY);
			
			IF TMR32.Q THEN
				ID3_Drive := FALSE;
				INPUT_VAR.ACTIVE_ID:=4;
				TMR30(IN:=FALSE);
				TMR31(IN:=FALSE);
				TMR32(IN:=FALSE);
			END_IF
		END_IF
	END_IF
4:
		IF STEP_DATA_4 = 0 THEN
			INPUT_VAR.ACTIVE_ID:=5;
		ELSE
			(*IF ID4_ALARM THEN
				Reset := TRUE;
				TMR40(IN:=TRUE,PT:= PROCESS_DELAY);
				IF TMR40.Q THEN
					Reset := FALSE;
				END_IF
			END_IF
			*)
			ID4_StepData :=STEP_DATA_4;
			TMR41(IN:=TRUE,PT:= PROCESS_DELAY);
			IF TMR41.Q THEN
				ID4_Drive := TRUE;
				TMR42(IN:=TMR41.Q,PT:= PROCESS_DELAY);
				
				IF TMR42.Q THEN
					ID4_Drive := FALSE;
					INPUT_VAR.ACTIVE_ID:=5;
					TMR40(IN:=FALSE);
					TMR41(IN:=FALSE);
					TMR42(IN:=FALSE);
				END_IF
			END_IF
		END_IF
	5:
		IF STEP_DATA_5 = 0 THEN
			INPUT_VAR.ACTIVE_ID:=0;
		ELSE
			(*
			IF ID5_ALARM THEN
				Reset := TRUE;
				TMR50(IN:=TRUE,PT:= PROCESS_DELAY);
				IF TMR50.Q THEN
					Reset := FALSE;
				END_IF
				
			END_IF
			*)
			ID5_StepData :=STEP_DATA_5;
			TMR51(IN:=TRUE,PT:= PROCESS_DELAY);
			IF TMR51.Q THEN
				ID5_Drive := TRUE;	
				TMR52(IN:=TMR51.Q,PT:= PROCESS_DELAY);
				IF TMR52.Q THEN
					ID5_Drive := FALSE;
					INPUT_VAR.ACTIVE_ID:=0;
					TMR50(IN:=FALSE);
					TMR51(IN:=FALSE);
					TMR52(IN:=FALSE);
			
				END_IF
			END_IF
		END_IF
		
END_CASE 

	//START_PROCESS := FALSE;
END_IF
TMR7(IN:=reset,PT:= T#1S);
IF  tmr7.Q THEN
	reset:=FALSE;
END_IF
IF ID1_ALARM OR ID2_ALARM OR ID3_ALARM OR ID4_ALARM OR ID5_ALARM THEN
			reset:=TRUE;
			ELSE
				reset:=FALSE;
			END_IF
IF reset THEN
	ID1_Reset := TRUE;
	ID2_Reset := TRUE;
	ID3_Reset := TRUE;
	ID4_Reset := TRUE;
	ID5_Reset := TRUE;
ELSE
	ID1_Reset := FALSE;
	ID2_Reset := FALSE;
	ID3_Reset := FALSE;
	ID4_Reset := FALSE;
	ID5_Reset := FALSE;
END_IF

END_PROGRAM

// ---- POUs/FUKUDA/RETURN_FUKUDA_1.TcPOU
PROGRAM RETURN_FUKUDA_1
VAR
END_VAR

CASE INPUT_VAR.I_CASE OF
0:
	IF INPUT_VAR.ACTIVE_ID=6 THEN
		INPUT_VAR.ACTIVE_ID:=1;
	END_IF
//	FUKUDA_MOVE(STEP_DATA_1:=0,STEP_DATA_2:=0,STEP_DATA_3:=0,STEP_DATA_4:=0,STEP_DATA_5:=2);
	CASE INPUT_VAR.I_CURRENT_TRANSACTION.TRANSPORT_INDEX OF
		2 : FUKUDA_MOVE(STEP_DATA_1:=3,
				STEP_DATA_2:=0,
				STEP_DATA_3:=3,
				STEP_DATA_4:=0,//2, //2
				STEP_DATA_5:=1);

		1 : FUKUDA_MOVE(STEP_DATA_1:=3,
				STEP_DATA_2:=0,
				STEP_DATA_3:=3,
				STEP_DATA_4:=1,//2, //2
				STEP_DATA_5:=0);
	END_CASE
1:
	IF INPUT_VAR.ACTIVE_ID=6 THEN
		INPUT_VAR.ACTIVE_ID:=1;
	END_IF
	
//	FUKUDA_MOVE(STEP_DATA_1:=6,STEP_DATA_2:=1,STEP_DATA_3:=21,STEP_DATA_4:=0,STEP_DATA_5:=0);
	FUKUDA_MOVE(STEP_DATA_1:=3,
				STEP_DATA_2:=0,
				STEP_DATA_3:=3,
				STEP_DATA_4:=0,
				STEP_DATA_5:=0);

2:
	IF INPUT_VAR.ACTIVE_ID=6 THEN
		INPUT_VAR.ACTIVE_ID:=1;
	END_IF
	
//	FUKUDA_MOVE(STEP_DATA_1:=6,STEP_DATA_2:=1,STEP_DATA_3:=21,STEP_DATA_4:=0,STEP_DATA_5:=0);
	FUKUDA_MOVE(STEP_DATA_1:=3,
				STEP_DATA_2:=0,
				STEP_DATA_3:=3,
				STEP_DATA_4:=0,
				STEP_DATA_5:=0);

3:
	IF INPUT_VAR.ACTIVE_ID=6 THEN
		INPUT_VAR.ACTIVE_ID:=1;
	END_IF
	
//	FUKUDA_MOVE(STEP_DATA_1:=6,STEP_DATA_2:=2,STEP_DATA_3:=21,STEP_DATA_4:=0,STEP_DATA_5:=0);
	FUKUDA_MOVE(STEP_DATA_1:=INPUT_VAR.I_CURRENT_TRANSACTION.TRANSPORT_INDEX+4,
				STEP_DATA_2:=1,
				STEP_DATA_3:=21,
				STEP_DATA_4:=0,
				STEP_DATA_5:=0);

4:
	IF INPUT_VAR.ACTIVE_ID=6 THEN
		INPUT_VAR.ACTIVE_ID:=1;
	END_IF
	
//	FUKUDA_MOVE(STEP_DATA_1:=6,STEP_DATA_2:=2,STEP_DATA_3:=21,STEP_DATA_4:=0,STEP_DATA_5:=0);
	FUKUDA_MOVE(STEP_DATA_1:=INPUT_VAR.I_CURRENT_TRANSACTION.TRANSPORT_INDEX+4,
				STEP_DATA_2:=1,
				STEP_DATA_3:=21,
				STEP_DATA_4:=0,
				STEP_DATA_5:=0);

5:
	IF INPUT_VAR.ACTIVE_ID=6 THEN
		INPUT_VAR.ACTIVE_ID:=1;
	END_IF
	
//	FUKUDA_MOVE(STEP_DATA_1:=6,STEP_DATA_2:=2,STEP_DATA_3:=21,STEP_DATA_4:=0,STEP_DATA_5:=0);
	FUKUDA_MOVE(STEP_DATA_1:=INPUT_VAR.I_CURRENT_TRANSACTION.TRANSPORT_INDEX+4,
				STEP_DATA_2:=2,
				STEP_DATA_3:=21,
				STEP_DATA_4:=0,
				STEP_DATA_5:=);
6:
	IF INPUT_VAR.ACTIVE_ID=6 THEN
		INPUT_VAR.ACTIVE_ID:=1;
	END_IF
	
//	FUKUDA_MOVE(STEP_DATA_1:=6,STEP_DATA_2:=2,STEP_DATA_3:=21,STEP_DATA_4:=0,STEP_DATA_5:=0);
	FUKUDA_MOVE(STEP_DATA_1:=INPUT_VAR.I_CURRENT_TRANSACTION.TRANSPORT_INDEX+4,
				STEP_DATA_2:=2,
				STEP_DATA_3:=2,
				STEP_DATA_4:=0,
				STEP_DATA_5:=0);
	input_var.o_CARTESSIAN_GRIPPER_ON:=TRUE;
	input_var.o_CARTESSIAN_GRIPPER_Off:=FALSE;
7:
	IF INPUT_VAR.ACTIVE_ID=6 THEN
		INPUT_VAR.ACTIVE_ID:=1;
	END_IF
	
	//	FUKUDA_MOVE(STEP_DATA_1:=1,STEP_DATA_2:=2,STEP_DATA_3:=3,STEP_DATA_4:=0,STEP_DATA_5:=0);
	FUKUDA_MOVE(STEP_DATA_1:=INPUT_VAR.I_CURRENT_TRANSACTION.STATION_NUMBER_LOAD,
				STEP_DATA_2:=2,
				STEP_DATA_3:=INPUT_VAR.I_CURRENT_TRANSACTION.JIG_INDEX_LOAD+4,
				STEP_DATA_4:=0,
				STEP_DATA_5:=0);

8:
	IF INPUT_VAR.ACTIVE_ID=6 THEN
		INPUT_VAR.ACTIVE_ID:=1;
	END_IF
//	FUKUDA_MOVE(STEP_DATA_1:=1,STEP_DATA_2:=4,STEP_DATA_3:=13,STEP_DATA_4:=0,STEP_DATA_5:=0);
	FUKUDA_MOVE(STEP_DATA_1:=INPUT_VAR.I_CURRENT_TRANSACTION.STATION_NUMBER_LOAD,
				STEP_DATA_2:=3,
				STEP_DATA_3:=INPUT_VAR.I_CURRENT_TRANSACTION.JIG_INDEX_LOAD+10,
				STEP_DATA_4:=0,
				STEP_DATA_5:=0);

9: 
	IF INPUT_VAR.ACTIVE_ID=6 THEN
		INPUT_VAR.ACTIVE_ID:=1;
	END_IF
	
//	FUKUDA_MOVE(STEP_DATA_1:=1,STEP_DATA_2:=3,STEP_DATA_3:=3,STEP_DATA_4:=0,STEP_DATA_5:=0);
	FUKUDA_MOVE(STEP_DATA_1:=INPUT_VAR.I_CURRENT_TRANSACTION.STATION_NUMBER_LOAD,
				STEP_DATA_2:=3,
				STEP_DATA_3:=INPUT_VAR.I_CURRENT_TRANSACTION.JIG_INDEX_LOAD+10,
				STEP_DATA_4:=0,
				STEP_DATA_5:=0);
10: 
	IF INPUT_VAR.ACTIVE_ID=6 THEN
		INPUT_VAR.ACTIVE_ID:=1;
	END_IF
	
//	FUKUDA_MOVE(STEP_DATA_1:=1,STEP_DATA_2:=3,STEP_DATA_3:=3,STEP_DATA_4:=0,STEP_DATA_5:=0);
	FUKUDA_MOVE(STEP_DATA_1:=INPUT_VAR.I_CURRENT_TRANSACTION.STATION_NUMBER_LOAD,
				STEP_DATA_2:=3,
				STEP_DATA_3:=INPUT_VAR.I_CURRENT_TRANSACTION.JIG_INDEX_LOAD+10,
				STEP_DATA_4:=0,
				STEP_DATA_5:=0);
11:
	IF INPUT_VAR.ACTIVE_ID=6 THEN
		INPUT_VAR.ACTIVE_ID:=1;
	END_IF
//	FUKUDA_MOVE(STEP_DATA_1:=1,STEP_DATA_2:=3,STEP_DATA_3:=13,STEP_DATA_4:=0,STEP_DATA_5:=0);
	FUKUDA_MOVE(STEP_DATA_1:=INPUT_VAR.I_CURRENT_TRANSACTION.STATION_NUMBER_LOAD,
				STEP_DATA_2:=4,
				STEP_DATA_3:=INPUT_VAR.I_CURRENT_TRANSACTION.JIG_INDEX_LOAD,
				STEP_DATA_4:=0,
				STEP_DATA_5:=0);

	input_var.o_CARTESSIAN_GRIPPER_ON:=FALSE;
	input_var.o_CARTESSIAN_GRIPPER_Off:=TRUE;
12: 
	
	IF INPUT_VAR.ACTIVE_ID=6 THEN
		INPUT_VAR.ACTIVE_ID:=1;
	END_IF
//	FUKUDA_MOVE(STEP_DATA_1:=1,STEP_DATA_2:=4,STEP_DATA_3:=3,STEP_DATA_4:=0,STEP_DATA_5:=0);
	FUKUDA_MOVE(STEP_DATA_1:=INPUT_VAR.I_CURRENT_TRANSACTION.STATION_NUMBER_LOAD,
				STEP_DATA_2:=3,
				STEP_DATA_3:=INPUT_VAR.I_CURRENT_TRANSACTION.JIG_INDEX_LOAD,
				STEP_DATA_4:=0,
				STEP_DATA_5:=0);
13: 
	
	IF INPUT_VAR.ACTIVE_ID=6 THEN
		INPUT_VAR.ACTIVE_ID:=1;
	END_IF
//	FUKUDA_MOVE(STEP_DATA_1:=1,STEP_DATA_2:=4,STEP_DATA_3:=3,STEP_DATA_4:=0,STEP_DATA_5:=0);
	FUKUDA_MOVE(STEP_DATA_1:=INPUT_VAR.I_CURRENT_TRANSACTION.STATION_NUMBER_LOAD,
				STEP_DATA_2:=3,
				STEP_DATA_3:=INPUT_VAR.I_CURRENT_TRANSACTION.JIG_INDEX_LOAD,
				STEP_DATA_4:=0,
				STEP_DATA_5:=0);

14: 
	
	IF INPUT_VAR.ACTIVE_ID=6 THEN
		INPUT_VAR.ACTIVE_ID:=1;
	END_IF
//	FUKUDA_MOVE(STEP_DATA_1:=1,STEP_DATA_2:=4,STEP_DATA_3:=3,STEP_DATA_4:=0,STEP_DATA_5:=0);
	FUKUDA_MOVE(STEP_DATA_1:=INPUT_VAR.I_CURRENT_TRANSACTION.STATION_NUMBER_LOAD,
				STEP_DATA_2:=4,
				STEP_DATA_3:=INPUT_VAR.I_CURRENT_TRANSACTION.JIG_INDEX_LOAD,
				STEP_DATA_4:=0,
				STEP_DATA_5:=0);

15:
	
	IF INPUT_VAR.ACTIVE_ID=6 THEN
		INPUT_VAR.ACTIVE_ID:=1;
	END_IF
	
//	FUKUDA_MOVE(STEP_DATA_1:=0,STEP_DATA_2:=1,STEP_DATA_3:=0,STEP_DATA_4:=0,STEP_DATA_5:=0);
	FUKUDA_MOVE(STEP_DATA_1:=0,
				STEP_DATA_2:=1,
				STEP_DATA_3:=0,
				STEP_DATA_4:=0,
				STEP_DATA_5:=0);

	END_CASE

END_PROGRAM

// ---- POUs/LASER/POU.TcPOU
PROGRAM POU
VAR
END_VAR

// NETWORK 1

END_PROGRAM

// ---- POUs/LOADER/STR.TcPOU
 PROGRAM STR
VAR

	NEW: INT;
	FG: INT;
	ENABLE_TIMER: BOOL := TRUE;
	TMR1: TON;
	TMR2: TON;
	CNT1: CTU;
	RST_COUNTER: BOOL;
END_VAR

ENABLE_TIMER:=INPUT_VAR.STRAIGHTEN_START;
IF ENABLE_TIMER THEN
	TMR1(IN:=NOT TMR2.Q,PT:=T#0.07S);
	TMR2(IN:=TMR1.Q,PT:=T#0.15S);
	IF TMR2.Q THEN
		TMR1(IN:=FALSE); 
		TMR2(IN:=FALSE);
	END_IF
	
	IF NOT  INDEXING_1_VAR.I_PRESS_STOPPER_DOWN  THEN
		INDEXING_1_VAR.O_PRESS_STOPPER_DOWN:=TRUE;
		INDEXING_1_VAR.O_PRESS_STOPPER_UP:=FALSE;
	END_IF
ELSE
		TMR1(IN:=FALSE);
		TMR2(IN:=FALSE);
END_IF
RST_COUNTER:=NOT ENABLE_TIMER;
CNT1(CU:=TMR1.Q,RESET:=RST_COUNTER,PV:=5);
IF CNT1.CV >=10 THEN
	ENABLE_TIMER:=FALSE;
	RST_COUNTER:=TRUE;
	INPUT_VAR.STRAIGHTEN_START:=FALSE;
	INDEXING_1_VAR.STRAIGHTEN_FINISH:=TRUE;
	INDEXING_1_VAR.O_PRESS_STOPPER_DOWN:=FALSE;
	INDEXING_1_VAR.O_PRESS_STOPPER_UP:=TRUE;
END_IF

IF CNT1.CV =2 THEN
	INDEXING_1_VAR.STRAIGHTEN_FINISH:=FALSE;
END_IF

IF 	INDEXING_1_VAR.STRAIGHTEN_FINISH THEN
	IF INDEXING_1_VAR.I_PRESS_STOPPER_UP THEN
		INPUT_VAR.STRAIGHTEN_DONE :=TRUE;	
		INPUT_VAR.STRAIGHTEN_PROCESS:=FALSE;
	END_IF	
END_IF
CASE CNT1.CV OF	
//CASE INDEXING_1_VAR.INDEXING_1_CASE OF
0:	
	INDEXING_1_VAR.O_PRESS_STOPPER_DOWN:=FALSE;
	INDEXING_1_VAR.O_PRESS_STOPPER_UP:=TRUE;
	//INDEXING_1_VAR.I_INDEXING_1_ROTATION_DONE:=FALSE;
	INDEXING_1_VAR.I_INDEXING_1_READY_FOR_STRAIGHTEN:=FALSE;
1:	
	INPUT_VAR.STRAIGHTEN_PROCESS:=TRUE;
	INDEXING_1_VAR.O_INDEXING_1_GRIPPER_OPEN_1:=TRUE;
	INDEXING_1_VAR.O_INDEXING_1_GRIPPER_CLOSE_1:=FALSE;
		
2:
	INDEXING_1_VAR.O_INDEXING_1_GRIPPER_EXT_UP :=TRUE;	
	INDEXING_1_VAR.O_INDEXING_1_GRIPPER_EXT_down:=FALSE;
	
3:
	INDEXING_1_VAR.O_INDEXING_1_GRIPPER_OPEN_1:=FALSE;
	INDEXING_1_VAR.O_INDEXING_1_GRIPPER_CLOSE_1:=TRUE;
			
4:
	INDEXING_1_VAR.O_INDEXING_1_GRIPPER_EXT_UP :=FALSE;	
	INDEXING_1_VAR.O_INDEXING_1_GRIPPER_EXT_down:=TRUE;

5:	
	INDEXING_1_VAR.O_INDEXING_1_GRIPPER_OPEN_1:=TRUE;
	INDEXING_1_VAR.O_INDEXING_1_GRIPPER_CLOSE_1:=FALSE;
		
6:
	INDEXING_1_VAR.O_INDEXING_1_GRIPPER_EXT_UP :=TRUE;	
	INDEXING_1_VAR.O_INDEXING_1_GRIPPER_EXT_down:=FALSE;	
7:
	INDEXING_1_VAR.O_INDEXING_1_GRIPPER_OPEN_1:=FALSE;
	INDEXING_1_VAR.O_INDEXING_1_GRIPPER_CLOSE_1:=TRUE;
			
8:
	INDEXING_1_VAR.O_INDEXING_1_GRIPPER_EXT_UP :=FALSE;	
	INDEXING_1_VAR.O_INDEXING_1_GRIPPER_EXT_down:=TRUE;

END_CASE

IF 
	INDEXING_1_VAR.O_INDEXING_1_GRIPPER_OPEN_1 AND
	INDEXING_1_VAR.I_INDEXING_1_GRIPPER_OPEN_1 AND
	INDEXING_1_VAR.I_INDEXING_1_GRIPPER_OPEN_2	AND
	INDEXING_1_VAR.I_INDEXING_1_GRIPPER_OPEN_3	AND 
	INDEXING_1_VAR.I_INDEXING_1_GRIPPER_OPEN_4	AND
	NOT INDEXING_1_VAR.I_INDEXING_1_GRIPPER_CLOSE_1	AND
	NOT INDEXING_1_VAR.I_INDEXING_1_GRIPPER_CLOSE_2	AND
	NOT INDEXING_1_VAR.I_INDEXING_1_GRIPPER_CLOSE_3	AND
	NOT INDEXING_1_VAR.I_INDEXING_1_GRIPPER_CLOSE_4 THEN
		INDEXING_1_VAR.I_ALL_GRIPPER_OPEN :=TRUE;
	END_IF

IF 
	NOT INDEXING_1_VAR.O_INDEXING_1_GRIPPER_OPEN_1 AND
	NOT INDEXING_1_VAR.I_INDEXING_1_GRIPPER_OPEN_1 AND
	NOT INDEXING_1_VAR.I_INDEXING_1_GRIPPER_OPEN_2	AND
	NOT INDEXING_1_VAR.I_INDEXING_1_GRIPPER_OPEN_3	AND 
	NOT INDEXING_1_VAR.I_INDEXING_1_GRIPPER_OPEN_4	AND
	INDEXING_1_VAR.I_INDEXING_1_GRIPPER_CLOSE_1	AND
	INDEXING_1_VAR.I_INDEXING_1_GRIPPER_CLOSE_2	AND
	INDEXING_1_VAR.I_INDEXING_1_GRIPPER_CLOSE_3	AND
	INDEXING_1_VAR.I_INDEXING_1_GRIPPER_CLOSE_4 THEN
		INDEXING_1_VAR.I_ALL_GRIPPER_OPEN :=FALSE;
END_IF


	INDEXING_1_VAR.O_INDEXING_1_GRIPPER_OPEN_2:=INDEXING_1_VAR.O_INDEXING_1_GRIPPER_OPEN_1;
	INDEXING_1_VAR.O_INDEXING_1_GRIPPER_OPEN_3:=INDEXING_1_VAR.O_INDEXING_1_GRIPPER_OPEN_1;
	INDEXING_1_VAR.O_INDEXING_1_GRIPPER_OPEN_4:=INDEXING_1_VAR.O_INDEXING_1_GRIPPER_OPEN_1;

	INDEXING_1_VAR.O_INDEXING_1_GRIPPER_CLOSE_2:=INDEXING_1_VAR.O_INDEXING_1_GRIPPER_CLOSE_1;
	INDEXING_1_VAR.O_INDEXING_1_GRIPPER_CLOSE_3:=INDEXING_1_VAR.O_INDEXING_1_GRIPPER_CLOSE_1;
	INDEXING_1_VAR.O_INDEXING_1_GRIPPER_CLOSE_4:=INDEXING_1_VAR.O_INDEXING_1_GRIPPER_CLOSE_1;

END_PROGRAM

// ---- POUs/ROBOT/INPUT_G61.TcPOU
PROGRAM INPUT_G61
VAR
(*	
ROBOT_I_GRIPPER_1 AT %IX100.0 : BOOL;
	ROBOT_I_GRIPPER_2 AT %IX100.1 : BOOL;
	ROBOT_I_GRIPPER_3 AT %IX100.2 : BOOL;
	ROBOT_I_GRIPPER_4 AT %IX100.3 : BOOL;
	
	ROBOT_I_GRIPPER_EXT_1 AT %IX100.4 : BOOL;
	ROBOT_I_GRIPPER_EXT_2 AT %IX100.5 : BOOL;
	ROBOT_I_GRIPPER_EXT_3 AT %IX100.6 : BOOL;
	ROBOT_I_GRIPPER_EXT_4 AT %IX100.7 : BOOL;
	
	ROBOT_O_GRIPPER_1 AT %IX101.0 : BOOL;
	ROBOT_O_GRIPPER_2 AT %IX101.1 : BOOL;
	ROBOT_O_GRIPPER_3 AT %IX101.2 : BOOL;
	ROBOT_O_GRIPPER_4 AT %IX101.3 : BOOL;
		
	ROBOT_O_GRIPPER_EXT_1 AT %IX101.4 : BOOL;
	ROBOT_O_GRIPPER_EXT_2 AT %IX101.5 : BOOL;
	ROBOT_O_GRIPPER_EXT_3 AT %IX101.6 : BOOL;
	ROBOT_O_GRIPPER_EXT_4 AT %IX101.7 : BOOL;
	
	*)
	TMR11: TON;
	TMR12: TON;
	TMR10: TON;
	TMR8: TON;
	TMR9: TON;
	TMR7: TON;
	TMR3: TON;
	TP1: TP;
	TMR1: TON;
	START_ROBOT: TP;
	TP2: TP;
	O_G6_HANG: BOOL;
	I_G6_HANG: BOOL;
	TMR2: TON;
	GO_ROBOT: BOOL;
	TP3: TP;
	TMR4: TON;
	CNT_CYCLE: CTU;
	START_ROTATE: R_TRIG;
	IN: INT;
END_VAR

IF INPUT_G6_VAR.I_G6_ENABLE  THEN
//GRIPPING 
IF INPUT_G6_VAR.IX_G6_GRIPPER_1 THEN
	INPUT_G6_VAR.O_G6_GRIPPER_CLOSE_1:=TRUE;
	INPUT_G6_VAR.O_G6_GRIPPER_OPEN_1:=FALSE;
ELSE
	INPUT_G6_VAR.O_G6_GRIPPER_CLOSE_1:=FALSE;
	INPUT_G6_VAR.O_G6_GRIPPER_OPEN_1:=TRUE;
END_IF

IF INPUT_G6_VAR.IX_G6_GRIPPER_2 THEN
	INPUT_G6_VAR.O_G6_GRIPPER_CLOSE_2:=TRUE;
	INPUT_G6_VAR.O_G6_GRIPPER_OPEN_2:=FALSE;
ELSE
	INPUT_G6_VAR.O_G6_GRIPPER_CLOSE_2:=FALSE;
	INPUT_G6_VAR.O_G6_GRIPPER_OPEN_2:=TRUE;
END_IF 

IF INPUT_G6_VAR.IX_G6_GRIPPER_3 THEN
	INPUT_G6_VAR.O_G6_GRIPPER_CLOSE_3:=TRUE;
	INPUT_G6_VAR.O_G6_GRIPPER_OPEN_3:=FALSE;
ELSE
	INPUT_G6_VAR.O_G6_GRIPPER_CLOSE_3:=FALSE;
	INPUT_G6_VAR.O_G6_GRIPPER_OPEN_3:=TRUE;
END_IF

IF INPUT_G6_VAR.IX_G6_GRIPPER_4 THEN
	INPUT_G6_VAR.O_G6_GRIPPER_CLOSE_4:=TRUE;
	INPUT_G6_VAR.O_G6_GRIPPER_OPEN_4:=FALSE;
ELSE
	INPUT_G6_VAR.O_G6_GRIPPER_CLOSE_4:=FALSE;
	INPUT_G6_VAR.O_G6_GRIPPER_OPEN_4:=TRUE;
END_IF

//EXTENDER DOWN
IF INPUT_G6_VAR.IX_G6_GRIPPER_EXT_1 THEN
	INPUT_G6_VAR.O_G6_GRIPPER_EXT_DOWN_1:=TRUE;
	INPUT_G6_VAR.O_G6_GRIPPER_EXT_UP_1:=FALSE;
ELSE
	INPUT_G6_VAR.O_G6_GRIPPER_EXT_DOWN_1:=FALSE;
	INPUT_G6_VAR.O_G6_GRIPPER_EXT_UP_1:=TRUE;
END_IF

IF INPUT_G6_VAR.IX_G6_GRIPPER_EXT_2 THEN
	INPUT_G6_VAR.O_G6_GRIPPER_EXT_DOWN_2:=TRUE;
	INPUT_G6_VAR.O_G6_GRIPPER_EXT_UP_2:=FALSE;
ELSE
	INPUT_G6_VAR.O_G6_GRIPPER_EXT_DOWN_2:=FALSE;
	INPUT_G6_VAR.O_G6_GRIPPER_EXT_UP_2:=TRUE;
END_IF

IF INPUT_G6_VAR.IX_G6_GRIPPER_EXT_3 THEN
	INPUT_G6_VAR.O_G6_GRIPPER_EXT_DOWN_3:=TRUE;
	INPUT_G6_VAR.O_G6_GRIPPER_EXT_UP_3:=FALSE;
ELSE
	INPUT_G6_VAR.O_G6_GRIPPER_EXT_DOWN_3:=FALSE;
	INPUT_G6_VAR.O_G6_GRIPPER_EXT_UP_3:=TRUE;
END_IF

IF INPUT_G6_VAR.IX_G6_GRIPPER_EXT_4 THEN
	INPUT_G6_VAR.O_G6_GRIPPER_EXT_DOWN_4:=TRUE;
	INPUT_G6_VAR.O_G6_GRIPPER_EXT_UP_4:=FALSE;
ELSE
	INPUT_G6_VAR.O_G6_GRIPPER_EXT_DOWN_4:=FALSE;
	INPUT_G6_VAR.O_G6_GRIPPER_EXT_UP_4:=TRUE;
END_IF





IF INPUT_VAR.ACTIVE_PROGRAM=2 THEN
	 INPUT_G6_VAR.O_G6_SELECT_FUKUDA_A:=TRUE;
ELSE
	INPUT_G6_VAR.O_G6_SELECT_FUKUDA_A:=FALSE;
END_IF

INPUT_VAR.I_STOPPER_TRANSFER_ON_A:= INPUT_VAR.O_STOPPER_TRANSFER_A;
IF INPUT_VAR.I_STOPPER_TRANSFER_ON_A OR INPUT_VAR.I_STOPPER_TRANSFER_ON_B THEN

INPUT_G6_VAR.O_G6_SETMOTORON:=TRUE;
TMR1(IN:=INPUT_G6_VAR.O_G6_SETMOTORON ,PT:=T#0.5S);
IF TMR1.Q THEN
	TP2(IN:=TMR1.Q,PT:=T#1S);
	INPUT_G6_VAR.O_G6_STOP:=TP2.Q;
	IF INPUT_G6_VAR.I_G6_READY THEN
		TP3(IN:=INPUT_G6_VAR.O_G6_SETMOTORON,PT:=T#0.1S);
		INPUT_G6_VAR.O_G6_HOME:=TP3.Q;
	END_IF
END_IF

IF INPUT_G6_VAR.O_G6_SETMOTORON AND INDEXING_1_VAR.I_INDEXING_1_ROTATION_DONE AND INDEXING_1_VAR.I_INDEXING_1_HOME THEN
	IF INPUT_G6_VAR.I_G6_READY OR INPUT_G6_VAR.I_G6_RUNNING THEN

// ERROR OVERRIDE
		IF 	INPUT_G6_VAR.I_G6_ERROR THEN
			TMR10(IN:=INPUT_G6_VAR.I_G6_ERROR,PT:=T#0.5S);
			IF NOT TMR10.Q THEN
				INPUT_G6_VAR.O_G6_RESET :=TRUE;	
				INPUT_G6_VAR.O_G6_START :=FALSE ;
				INPUT_G6_VAR.O_G6_CONTINUE :=FALSE;
			ELSE
				INPUT_G6_VAR.O_G6_RESET :=FALSE;		
			END_IF
		END_IF
	 
		//TMR8(IN:=INPUT_G6_VAR.O_G6_SELECT_FUKUDA_A,PT:=T#5S);
		//TMR9(IN:=INPUT_G6_VAR.O_G6_START,PT:=T#2S);
		
//START FOR 1ST TIME
		IF INPUT_G6_VAR.I_G6_READY AND NOT INPUT_G6_VAR.I_G6_ERROR AND NOT INPUT_G6_VAR.I_G6_RUNNING THEN
			TMR7(IN:=INPUT_G6_VAR.I_G6_READY,PT:=T#1S);
			START_ROBOT(IN:=TMR7.Q,PT:=T#2S);
			INPUT_G6_VAR.O_G6_START :=TMR7.Q ;
			INPUT_G6_VAR.O_G6_STOP:=FALSE;
		ELSE
			TMR7(IN:=FALSE);
		END_IF
		IF  NOT INPUT_G6_VAR.I_G6_READY THEN
			INPUT_G6_VAR.O_G6_START :=FALSE ;
		END_IF
		
//STOP 
		IF INPUT_G6_VAR.I_G6_END_FUKUDA AND NOT INPUT_G6_VAR.I_G6_READY AND NOT INPUT_G6_VAR.I_G6_RUNNING THEN
			TMR8(IN:=FALSE);
			TMR9(IN:=FALSE);
		//	INPUT_G6_VAR.O_G6_STOP:=TRUE;
		END_IF
		TMR2(IN:=INPUT_G6_VAR.O_G6_STOP,PT:=T#1S);
		IF TMR2.Q THEN
			INPUT_G6_VAR.I_G6_HANG:=FALSE;
			INPUT_G6_VAR.O_G6_STOP:=FALSE;
			TMR1(IN:=FALSE);
		END_IF
		
//CONTINUE	
		GO_ROBOT:=(INPUT_G6_VAR.I_G6_READY_PLACING  AND (LOADER_RS4_VAR.I_LOADER_RS4_READY_TAKEUP OR NOT LOADER_RS4_VAR.I_LOADER_RS4_ENABLE)  AND INDEXING_2_VAR.O_ROTATION_DONE );	
		IF INPUT_G6_VAR.I_G6_RUNNING AND  INDEXING_1_VAR.I_INDEXING_1_ROTATION_DONE AND GO_ROBOT AND INPUT_VAR.STRAIGHTEN_DONE AND NOT INPUT_G6_VAR.I_G6_END_FUKUDA AND INPUT_G6_VAR.I_G6_RUNNING AND NOT LOADER_RS4_VAR.I_LOADER_RS4_END_CARRIER THEN
				TMR3(IN:=GO_ROBOT ,PT:=T#0.5S);
				TP1(IN:=GO_ROBOT,PT:=T#0.1S);
		ELSE
			TMR3(IN:=FALSE);
			TP1(IN:=FALSE);
		END_IF
		INPUT_G6_VAR.O_G6_CONTINUE :=TMR3.Q;

//
		CNT_CYCLE(CU:=INPUT_G6_VAR.I_G6_START_TAKEUP,RESET:=INPUT_G6_VAR.I_G6_DISABLE,PV:=4);
		IF CNT_CYCLE.CV >=3 THEN
			LOADER_RS4_VAR.I_LOADER_RS4_ENABLE:=TRUE;
 		END_IF
		IF NOT LOADER_RS4_VAR.I_LOADER_RS4_ENABLE AND INPUT_G6_VAR.I_G6_END_CYCLE THEN
			START_ROTATE(CLK:=TRUE);
			//INDEXING_1_VAR.O_ROTATION_START:= START_ROTATE.Q;	
			ELSE
			START_ROTATE(CLK:=FALSE);
		END_IF

	END_IF
END_IF
END_IF

END_IF

END_PROGRAM
